# B&R Automation Studio project PrzewijarkaBRPraktyki
Automation Studio 4.12.8.41 SP; technology packages: mapp 5.24.5, mappCockpit 5.24.4, mappControl 5.24.2, mappMotion 5.29.0, mappView 5.24.5

## Configuration PrzewijarkaPraktykiBR

CPU X20CP0483, AutomationRuntime J4.93, Build 4.1.2, Safety 0.0, Vc V4.73.2

### Task classes (Cpu.sw)
```
Cyclic#4 (cycle 100000 us, tolerance 100000 us):
  PID <- Control.PID.PID.prg
  Tension <- Control.Tension.Tension.prg
  Axis1 <- Control.Axis.Axis1.Axis1.prg
  Axis2 <- Control.Axis.Axis2.Axis2.prg
  Axis3 <- Control.Axis.Axis3.Axis3.prg
  Axes <- Control.Axis.Axes.prg
  PackML <- PackMLCore.PackML.prg
NcDataObjects: mcdrivelog
Binaries: Settings, arcoal, mvLoader, arsvcreg, FWRules, arflatprv, udbdef, mCoWebSc, TCData, arconfig, User, sysconf, Role, iomap, asfw, ashwac, ashwd
Libraries: McBase, MpBase, sys_lib, arssl, MpAxis, McAxis, McAcpAx, MpAlarmX, astime, runtime, MpServer, CoTrace, AsZip, FileIO, MpRegMark, MpTension, MpPackML
```

### Hardware
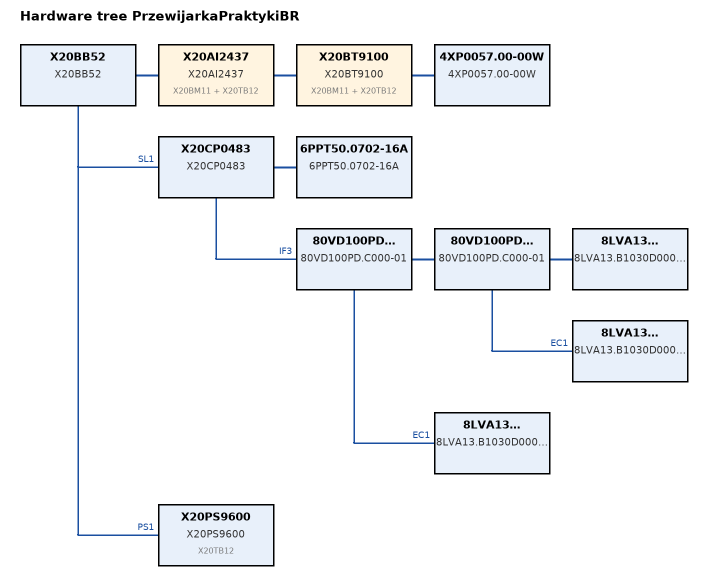
```
4XP0057.00-00W : 4XP0057.00-00W v2.1.0.0  [X2X1 -> X20BT9100.X2X1 [Cable Type=X2XCable, Length=10, Version=1.0.0.3]]
6PPT50.0702-16A : 6PPT50.0702-16A v1.3.8.0  [ETH1 -> X20CP0483.IF2 [Cable Type=PowerlinkCable, Length=10, Version=1.0.0.3]]
  Terminal = true
  Startmode = 2
  Mode = Manual
  InternetAddress = 192.168.0.12
  Subnetmask = 255.255.255.0
  PasswordVNC = 
  SelectedFavoriteWeb = 192.168.0.2
  Favorites_Web1 = webserver1
  PasswordCIFS = 
  PasswordService = 
80VD100PD.C000-01 : 80VD100PD.C000-01 v2.5.0.0  [PLK1 -> X20CP0483.IF3 (NodeNumber=1) [Cable Type=PowerlinkCable, Length=10, Version=1.0.0.3]; PLK2 -> 80VD100PD.C000-01a.PLK1 (NodeNumber=1) [Cable Type=PowerlinkCable, Length=10, Version=1.0.0.3]; EC1 -> 8LVA13.B1030D000-0.EC]
  DriveConfiguration/Module:
    McAcoposTypeID = AcoposMicroDConfig
    ActivateACOPOSSimulationOnPLC = 0
  DriveConfiguration/Channel[1]/RealAxis:
    AxisReference = gAxis_1
    MechanicalElementsIsInvisible = 0
  DriveConfiguration/Channel[1]/RealAxis/MechanicalElements/Gearbox:
    InputIsReadOnly = 0
    Input = 3
    OutputIsReadOnly = 0
    Output = 1
  DriveConfiguration/Channel[1]/RealAxis/MechanicalElements/RotaryToLinearTransformation:
    ReferenceDistanceIsReadOnly = 0
    ReferenceDistance = 360
  DriveConfiguration/Channel[1]/RealAxis/Controller:
    ModeIsReadOnly = 0
    Mode = PositionController
  DriveConfiguration/Channel[1]/RealAxis/Controller/Mode/Position:
    ProportionalGain = 358.000000
    IntegrationTime = 0.0
    PredictionTime = 0.0004
    TotalDelayTime = 0.0004
  DriveConfiguration/Channel[1]/RealAxis/Controller/Mode/Speed:
    ProportionalGainIsReadOnly = 0
    ProportionalGain = 1.150000
    IntegrationTimeIsReadOnly = 0
    IntegrationTime = 0.0
    FilterTimeIsReadOnly = 0
    FilterTime = 0.0
  DriveConfiguration/Channel[1]/RealAxis/Controller/Mode/LoopFilters:
    LoopFilterXIsReadOnly = 0
    LoopFilter1 = NotUsed
    LoopFilter2 = NotUsed
    LoopFilter3 = NotUsed
  DriveConfiguration/Channel[1]/RealAxis/Homing:
    ModeIsReadOnly = 0
    Mode = Direct
  DriveConfiguration/Channel[1]/RealAxis/Homing/Mode:
    Position = 0.0
    ReferencePulse = NotUsed
  DriveConfiguration/Channel[1]/RealAxis/Homing:
    RestorePositionVariable = 
  DriveConfiguration/Channel[1]/RealAxis/StopReaction:
    QuickstopIsReadOnly = 0
    Quickstop = DecelerationLimit
    DriveErrorIsReadOnly = 0
    DriveError = DecelerationLimit
    FilterTime = 0.0
  DriveConfiguration/Channel[1]/RealAxis/MovementErrorLimits:
    PositionError = 1.0
    VelocityErrorMonitoring = Automatic1
  DriveConfiguration/Channel[1]/RealAxis:
    JerkFilterIsReadOnly = 0
    JerkFilter = NotUsed
    ZeroVibrationFilter = NotUsed
  DriveConfiguration/Channel[1]/RealAxis/DigitalInputs/HomingSwitch:
    SourceIsReadOnly = 0
    Source = NotUsed
    Level = High
  DriveConfiguration/Channel[1]/RealAxis/DigitalInputs/PositiveLimitSwitch:
    SourceIsReadOnly = 0
    Source = NotUsed
    Level = High
  DriveConfiguration/Channel[1]/RealAxis/DigitalInputs/NegativeLimitSwitch:
    SourceIsReadOnly = 0
    Source = NotUsed
    Level = High
  DriveConfiguration/Channel[1]/RealAxis/DigitalInputs/Trigger1:
    Source = X2Trigger1
    Level = High
  DriveConfiguration/Channel[1]/RealAxis/DigitalInputs/Trigger2:
    Source = X2Trigger2
    Level = High
  DriveConfiguration/Channel[1]/RealAxis/DigitalInputs/Quickstop:
    Input = Trigger2
  DriveConfiguration/Channel[1]/RealAxis/Simulation:
    SimulationModeOnPLC = SetValueGeneration
    SimulationModeOnACOPOS = NotUsed
  DriveConfiguration/Channel[1]:
    ExternalEncoderAxis = NotUsed
  DriveConfiguration/Channel[2]/RealAxis:
    AxisReference = 
    MechanicalElementsIsInvisible = 0
  DriveConfiguration/Channel[2]/RealAxis/MechanicalElements/Gearbox:
    InputIsReadOnly = 0
    Input = 1
    OutputIsReadOnly = 0
    Output = 1
  DriveConfiguration/Channel[2]/RealAxis/MechanicalElements/RotaryToLinearTransformation:
    ReferenceDistanceIsReadOnly = 0
    ReferenceDistance = 1
  DriveConfiguration/Channel[2]/RealAxis/Controller:
    ModeIsReadOnly = 0
    Mode = PositionController
  DriveConfiguration/Channel[2]/RealAxis/Controller/Mode/Position:
    ProportionalGain = 50.0
    IntegrationTime = 0.0
    PredictionTime = 0.0004
    TotalDelayTime = 0.0004
  DriveConfiguration/Channel[2]/RealAxis/Controller/Mode/Speed:
    ProportionalGainIsReadOnly = 0
    ProportionalGain = 2.0
    IntegrationTimeIsReadOnly = 0
    IntegrationTime = 0.0
    FilterTimeIsReadOnly = 0
    FilterTime = 0.0
  DriveConfiguration/Channel[2]/RealAxis/Controller/Mode/LoopFilters:
    LoopFilterXIsReadOnly = 0
    LoopFilter1 = NotUsed
    LoopFilter2 = NotUsed
    LoopFilter3 = NotUsed
  DriveConfiguration/Channel[2]/RealAxis/Homing:
    ModeIsReadOnly = 0
    Mode = Direct
  DriveConfiguration/Channel[2]/RealAxis/Homing/Mode:
    Position = 0.0
    ReferencePulse = NotUsed
  DriveConfiguration/Channel[2]/RealAxis/Homing:
    RestorePositionVariable = 
  DriveConfiguration/Channel[2]/RealAxis/StopReaction:
    QuickstopIsReadOnly = 0
    Quickstop = DecelerationLimit
    DriveErrorIsReadOnly = 0
    DriveError = DecelerationLimit
    FilterTime = 0.0
  DriveConfiguration/Channel[2]/RealAxis/MovementErrorLimits:
    PositionError = 1.0
    VelocityErrorMonitoring = Automatic1
  DriveConfiguration/Channel[2]/RealAxis:
    JerkFilterIsReadOnly = 0
    JerkFilter = NotUsed
    ZeroVibrationFilter = NotUsed
  DriveConfiguration/Channel[2]/RealAxis/DigitalInputs/HomingSwitch:
    SourceIsReadOnly = 0
    Source = NotUsed
    Level = High
  DriveConfiguration/Channel[2]/RealAxis/DigitalInputs/PositiveLimitSwitch:
    SourceIsReadOnly = 0
    Source = NotUsed
    Level = High
  DriveConfiguration/Channel[2]/RealAxis/DigitalInputs/NegativeLimitSwitch:
    SourceIsReadOnly = 0
    Source = NotUsed
    Level = High
  DriveConfiguration/Channel[2]/RealAxis/DigitalInputs/Trigger1:
    Source = X2Trigger1
    Level = High
  DriveConfiguration/Channel[2]/RealAxis/DigitalInputs/Trigger2:
    Source = X2Trigger2
    Level = High
  DriveConfiguration/Channel[2]/RealAxis/DigitalInputs/Quickstop:
    Input = Trigger2
  DriveConfiguration/Channel[2]/RealAxis/Simulation:
    SimulationModeOnPLC = SetValueGeneration
    SimulationModeOnACOPOS = NotUsed
  DriveConfiguration/Channel[2]:
    ExternalEncoderAxis = NotUsed
80VD100PD.C000-01a : 80VD100PD.C000-01 v2.5.0.0  [PLK1 -> 80VD100PD.C000-01.PLK2 (NodeNumber=2) [Cable Type=PowerlinkCable, Length=10, Version=1.0.0.3]; EC1 -> 8LVA13.B1030D000-0b.EC; EC2 -> 8LVA13.B1030D000-0a.EC; MT2 -> 8LVA13.B1030D000-0a.MT]
  DriveConfiguration/Module:
    McAcoposTypeID = AcoposMicroDConfig
    ActivateACOPOSSimulationOnPLC = 0
  DriveConfiguration/Channel[1]/RealAxis:
    AxisReference = gAxis_2
    MechanicalElementsIsInvisible = 0
  DriveConfiguration/Channel[1]/RealAxis/MechanicalElements/Gearbox:
    InputIsReadOnly = 0
    Input = 3
    OutputIsReadOnly = 0
    Output = 1
  DriveConfiguration/Channel[1]/RealAxis/MechanicalElements/RotaryToLinearTransformation:
    ReferenceDistanceIsReadOnly = 0
    ReferenceDistance = 191.637
  DriveConfiguration/Channel[1]/RealAxis/Controller:
    ModeIsReadOnly = 0
    Mode = PositionController
  DriveConfiguration/Channel[1]/RealAxis/Controller/Mode/Position:
    ProportionalGain = 124.000000
    IntegrationTime = 0.0
    PredictionTime = 0.0004
    TotalDelayTime = 0.0004
  DriveConfiguration/Channel[1]/RealAxis/Controller/Mode/Speed:
    ProportionalGainIsReadOnly = 0
    ProportionalGain = 0.950000
    IntegrationTimeIsReadOnly = 0
    IntegrationTime = 0.0
    FilterTimeIsReadOnly = 0
    FilterTime = 0.0
  DriveConfiguration/Channel[1]/RealAxis/Controller/Mode/LoopFilters:
    LoopFilterXIsReadOnly = 0
    LoopFilter1 = NotUsed
    LoopFilter2 = NotUsed
    LoopFilter3 = NotUsed
  DriveConfiguration/Channel[1]/RealAxis/Homing:
    ModeIsReadOnly = 0
    Mode = Direct
  DriveConfiguration/Channel[1]/RealAxis/Homing/Mode:
    Position = 0.0
    ReferencePulse = NotUsed
  DriveConfiguration/Channel[1]/RealAxis/Homing:
    RestorePositionVariable = 
  DriveConfiguration/Channel[1]/RealAxis/StopReaction:
    QuickstopIsReadOnly = 0
    Quickstop = DecelerationLimit
    DriveErrorIsReadOnly = 0
    DriveError = DecelerationLimit
    FilterTime = 0.0
  DriveConfiguration/Channel[1]/RealAxis/MovementErrorLimits:
    PositionError = 1.0
    VelocityErrorMonitoring = Automatic1
  DriveConfiguration/Channel[1]/RealAxis:
    JerkFilterIsReadOnly = 0
    JerkFilter = NotUsed
    ZeroVibrationFilter = NotUsed
  DriveConfiguration/Channel[1]/RealAxis/DigitalInputs/HomingSwitch:
    SourceIsReadOnly = 0
    Source = NotUsed
    Level = High
  DriveConfiguration/Channel[1]/RealAxis/DigitalInputs/PositiveLimitSwitch:
    SourceIsReadOnly = 0
    Source = NotUsed
    Level = High
  DriveConfiguration/Channel[1]/RealAxis/DigitalInputs/NegativeLimitSwitch:
    SourceIsReadOnly = 0
    Source = NotUsed
    Level = High
  DriveConfiguration/Channel[1]/RealAxis/DigitalInputs/Trigger1:
    Source = X2Trigger1
    Level = High
  DriveConfiguration/Channel[1]/RealAxis/DigitalInputs/Trigger2:
    Source = X2Trigger2
    Level = High
  DriveConfiguration/Channel[1]/RealAxis/DigitalInputs/Quickstop:
    Input = Trigger2
  DriveConfiguration/Channel[1]/RealAxis/Simulation:
    SimulationModeOnPLC = SetValueGeneration
    SimulationModeOnACOPOS = NotUsed
  DriveConfiguration/Channel[1]:
    VirtualAxis = Used
  DriveConfiguration/Channel[1]/VirtualAxis:
    AxisReference = 
  DriveConfiguration/Channel[1]/VirtualAxis/Homing:
    Mode = Direct
  DriveConfiguration/Channel[1]/VirtualAxis/Homing/Mode:
    Position = 0.0
  DriveConfiguration/Channel[1]/VirtualAxis/Homing:
    RestorePositionVariable = 
  DriveConfiguration/Channel[1]/VirtualAxis:
    JerkFilterIsReadOnly = 0
    JerkFilter = NotUsed
    ZeroVibrationFilter = NotUsed
  DriveConfiguration/Channel[1]:
    ExternalEncoderAxis = NotUsed
  DriveConfiguration/Channel[2]/RealAxis:
    AxisReference = gAxis_3
    MechanicalElementsIsInvisible = 0
  DriveConfiguration/Channel[2]/RealAxis/MechanicalElements/Gearbox:
    InputIsReadOnly = 0
    Input = 3
    OutputIsReadOnly = 0
    Output = 1
  DriveConfiguration/Channel[2]/RealAxis/MechanicalElements/RotaryToLinearTransformation:
    ReferenceDistanceIsReadOnly = 0
    ReferenceDistance = 360
  DriveConfiguration/Channel[2]/RealAxis/Controller:
    ModeIsReadOnly = 0
    Mode = PositionController
  DriveConfiguration/Channel[2]/RealAxis/Controller/Mode/Position:
    ProportionalGain = 358
    IntegrationTime = 0.0
    PredictionTime = 0.0004
    TotalDelayTime = 0.0004
  DriveConfiguration/Channel[2]/RealAxis/Controller/Mode/Speed:
    ProportionalGainIsReadOnly = 0
    ProportionalGain = 1.15
    IntegrationTimeIsReadOnly = 0
    IntegrationTime = 0.0
    FilterTimeIsReadOnly = 0
    FilterTime = 0.0
  DriveConfiguration/Channel[2]/RealAxis/Controller/Mode/LoopFilters:
    LoopFilterXIsReadOnly = 0
    LoopFilter1 = NotUsed
    LoopFilter2 = NotUsed
    LoopFilter3 = NotUsed
  DriveConfiguration/Channel[2]/RealAxis/Homing:
    ModeIsReadOnly = 0
    Mode = Direct
  DriveConfiguration/Channel[2]/RealAxis/Homing/Mode:
    Position = 0.0
    ReferencePulse = NotUsed
  DriveConfiguration/Channel[2]/RealAxis/Homing:
    RestorePositionVariable = 
  DriveConfiguration/Channel[2]/RealAxis/StopReaction:
    QuickstopIsReadOnly = 0
    Quickstop = DecelerationLimit
    DriveErrorIsReadOnly = 0
    DriveError = DecelerationLimit
    FilterTime = 0.0
  DriveConfiguration/Channel[2]/RealAxis/MovementErrorLimits:
    PositionError = 1.0
    VelocityErrorMonitoring = Automatic1
  DriveConfiguration/Channel[2]/RealAxis:
    JerkFilterIsReadOnly = 0
    JerkFilter = NotUsed
    ZeroVibrationFilter = NotUsed
  DriveConfiguration/Channel[2]/RealAxis/DigitalInputs/HomingSwitch:
    SourceIsReadOnly = 0
    Source = NotUsed
    Level = High
  DriveConfiguration/Channel[2]/RealAxis/DigitalInputs/PositiveLimitSwitch:
    SourceIsReadOnly = 0
    Source = NotUsed
    Level = High
  DriveConfiguration/Channel[2]/RealAxis/DigitalInputs/NegativeLimitSwitch:
    SourceIsReadOnly = 0
    Source = NotUsed
    Level = High
  DriveConfiguration/Channel[2]/RealAxis/DigitalInputs/Trigger1:
    Source = X2Trigger1
    Level = High
  DriveConfiguration/Channel[2]/RealAxis/DigitalInputs/Trigger2:
    Source = X2Trigger2
    Level = High
  DriveConfiguration/Channel[2]/RealAxis/DigitalInputs/Quickstop:
    Input = Trigger2
  DriveConfiguration/Channel[2]/RealAxis/Simulation:
    SimulationModeOnPLC = SetValueGeneration
    SimulationModeOnACOPOS = NotUsed
  DriveConfiguration/Channel[2]:
    ExternalEncoderAxis = NotUsed
8LVA13.B1030D000-0 : 8LVA13.B1030D000-0 v2.2.0.3  [EC -> 80VD100PD.C000-01.EC1; MT -> 80VD100PD.C000-01.MT1]
  M1/MotorParameters:
    MOTOR_AMB_TEMP_RATED = 40
8LVA13.B1030D000-0a : 8LVA13.B1030D000-0 v2.2.0.3  [EC -> 80VD100PD.C000-01a.EC2; MT -> 80VD100PD.C000-01a.MT2]
  M1/MotorParameters:
    MOTOR_AMB_TEMP_RATED = 40
8LVA13.B1030D000-0b : 8LVA13.B1030D000-0 v2.2.0.3  [EC -> 80VD100PD.C000-01a.EC1; MT -> 80VD100PD.C000-01a.MT1]
  M1/MotorParameters:
    MOTOR_AMB_TEMP_RATED = 40
X20AI2437 : X20AI2437 v1.3.0.0  [SS1 -> X20TB12a.SS; SL -> X20BM11.SL1]
X20BB52 : X20BB52 v1.2.0.0
X20BM11 : X20BM11 v1.1.0.0  [X2X1 -> X20BB52.IF6]
X20BM11a : X20BM11 v1.1.0.0  [X2X1 -> X20BM11.X2X2]
X20BT9100 : X20BT9100 v1.3.0.0  [SS1 -> X20TB12b.SS; SL -> X20BM11a.SL1]
X20CP0483 : X20CP0483 v1.6.0.0  [SL -> X20BB52.SL1]
  Connector IF2:
    ActivateDevice = 1
    Mode = Manual
    InternetAddress = 192.168.0.2
    SubnetMask = 255.255.255.0
  Connector IF3:
    Channel1
    ChannelID1 = McAcpBroadcast
    ChannelType1 = OCTET[36]
  ConfigurationID = PrzewijarkaBRPraktyki_PrzewijarkaPraktykiBR
  TimerDeviceType = EPLX2X
  TimerDevice = X20CP0483.IF3
  TaskClassIdleTime = 2000
  Cyclic1Duration = 2000
  Cyclic1Tolerance = 0
  Cyclic1Stack = 30000
  Cyclic1Output = 1
  Cyclic2Duration = 20000
  Cyclic2Tolerance = 20000
  Cyclic3Duration = 50000
  Cyclic3Tolerance = 50000
  Cyclic4Duration = 100000
  Cyclic4Tolerance = 100000
  Cyclic5Duration = 200000
  Cyclic5Tolerance = 200000
  Cyclic6Duration = 500000
  Cyclic6Tolerance = 500000
  Cyclic7Duration = 1000000
  Cyclic7Tolerance = 1000000
  Cyclic8Duration = 10000
  Cyclic8Tolerance = 30000000
  FileDevice1
  FileDeviceName1 = USER
  FileDevicePath1 = USER_PATH
  FileDevice2
  FileDeviceName2 = RECIPE
  FileDevicePath2 = USER_PATH/Recipe
  FileDevice3
  FileDeviceName3 = DATA
  FileDevicePath3 = USER_PATH/Data
  TimeZone = 160
  ActivateDaylightSavingTime = 1
  ActivateSntpServer = 1
  EthernetDefaultGateway = 192.168.0.1
  FtpUser1
  FtpUsername1 = AdminFTP
  FtpUserPassword1 = 6YI7hPEHEUgPCGBGJ1BSV9dcZzKYXQvWVp6sNHSerZA=  // Admin123
  FtpUserSalt1 = /B0I6o9l
  FTPAccessRight1 = 0
  ActivateOpcUa = 1
  OpcUaInformationModels_PV_Version = 1
X20PS9600 : X20PS9600 v1.6.0.0  [PS -> X20BB52.PS1; SS1 -> X20TB12.SS]
X20TB12 : X20TB12 v1.0.0.0
X20TB12a : X20TB12 v1.0.0.0
X20TB12b : X20TB12 v1.0.0.0
```

### IoMap.iom - X20CP0483/IoMap.iom
```iecst
VAR_CONFIG
	::gHMI.ModuleOK.PowerSupply AT %IX."X20PS9600".ModuleOk;
	::gHMI.ModuleOK.AnalogInput AT %IX."X20AI2437".ModuleOk;
	::gHMI.ModuleOK.SystemBusTransmitter AT %IX."X20BT9100".ModuleOk;
	::gHMI.ModuleOK.ControlKeypad AT %IX."4XP0057.00-00W".ModuleOk;
	::Tension:ActRightDancerPos AT %IW."X20AI2437".AnalogInput01;
	::Tension:ActLeftDancerPos AT %IW."X20AI2437".AnalogInput02;
	::MainPage:PhysicalBtn.Production.Start.State AT %IX."4XP0057.00-00W".DigitalInput01;
	::MainPage:PhysicalBtn.Production.Stop.State AT %IX."4XP0057.00-00W".DigitalInput02;
	::MainPage:PhysicalBtn.Production.Reset.State AT %IX."4XP0057.00-00W".DigitalInput05;
	::MainPage:PhysicalBtn.Manual.Left.State AT %IX."4XP0057.00-00W".DigitalInput03;
	::MainPage:PhysicalBtn.Manual.Right.State AT %IX."4XP0057.00-00W".DigitalInput04;
	::MainPage:PhysicalBtn.Production.Start.ColorON AT %QX."4XP0057.00-00W".DigitalOutput01;
	::MainPage:PhysicalBtn.Production.Stop.ColorON AT %QX."4XP0057.00-00W".DigitalOutput07;
	::MainPage:PhysicalBtn.Manual.Left.ColorON AT %QX."4XP0057.00-00W".DigitalOutput12;
	::MainPage:PhysicalBtn.Manual.Right.ColorON AT %QX."4XP0057.00-00W".DigitalOutput16;
	::MainPage:PhysicalBtn.Production.Reset.ColorON AT %QX."4XP0057.00-00W".DigitalOutput20;
END_VAR
```

### Config_2.tensioncontroller - X20CP0483/mappControl/Config_2.tensioncontroller
```
Element gTensionCtrl_Unwinder (Type=tensioncontroller)  // axis1
  TensionController:
    MotionSystem = mappMotion
      AxisReference = gAxis_1
      AxisVelocityProfile:
        Acceleration = 0.5
        Deceleration = 0.5
        StopDeceleration = 2
    Utilization:
      Winder:
        MinimumDiameter = 30
        MaximumDiameter = 80
    Controller:
      PIDParameters:
        OperatingPoint[1]
      MaximumVelocityCorrection = 1
      ToleranceBand:
        Lower = 4
        Upper = 4
      Initialization:
        MaximumLineVelocityCorrection = 1
    Material:
      Length = 0.4
      Width = 48
      TensionLimit = 300
    InputSignals:
      SetMaterialTension = 
Element gTensionCtrl_Rewinder (Type=tensioncontroller)  // axis3
  TensionController:
    MotionSystem = mappMotion
      AxisReference = gAxis_3
      AxisVelocityProfile:
        Acceleration = 0.5
        Deceleration = 0.5
        StopDeceleration = 2
    Utilization = Rewind
      Winder:
        MinimumDiameter = 30
        MaximumDiameter = 80
    Controller:
      PIDParameters:
        OperatingPoint[1]
      ToleranceBand:
        Lower = 4
        Upper = 4
      Initialization:
        MaximumLineVelocityCorrection = 1
    Material:
      Length = 0.4
      Width = 48
      TensionLimit = 300
    InputSignals:
      SetMaterialTension = 
Element gTensionCtrl_Master (Type=tensioncontroller)
  TensionController:
    Utilization = Transport
    Controller = Master
Element gTensionCtrl_TransportDancer (Type=tensioncontroller)  // axis2
  TensionController:
    MotionSystem = mappMotion
      AxisReference = gAxis_2
      AxisVelocityProfile:
        Acceleration = 0.5
        Deceleration = 0.5
        StopDeceleration = 2
    Utilization = Transport
    Controller = DancerControl
      PIDParameters:
        OperatingPoint[1]
      Orientation = 1
      Initialization:
        MaximumLineVelocityCorrection = 1
    Material:
      Length = 0.4
      TensionLimit = 300
    InputSignals:
      SetDancerPosition = 
Element gTensionCtrl_TransportTension (Type=tensioncontroller)
  TensionController:
    Utilization = Transport
    Controller:
      PIDParameters:
        OperatingPoint[1]
```

### Config_3.tensiongroup - X20CP0483/mappControl/Config_3.tensiongroup
```
Element gTensionGroup_1 (Type=tensiongroup)
  Linking:
    Subnodes:
      Zone[0] = gTensionCtrl_Unwinder
      Zone[1] = gTensionCtrl_TransportDancer
      Zone[2] = gTensionCtrl_Rewinder
  TensionGroup:
    Simulation = 1
    CommonZoneSettings:
      Material:
        Width = 48
        TensionLimit = 300
    InputSignals:
      GroupLineVelocity = ::Tension:TensionVar.GroupLineVelocity
    Features:
      FeatureRef[0] = 
```

### Config_4.regmarkdetection - X20CP0483/mappControl/Config_4.regmarkdetection
```
Element gRegMarkDetection_1 (Type=regmarkdetection)
  RegistrationMarkDetection:
    SensorSignal:
      AxisReference = gAxis_2
```

### Config_8.purevaxcfg - X20CP0483/mappMotion/Config_8.purevaxcfg
```
Element PureVAxCfg_1 (Type=purevaxcfg)
  TypeID = PureVAxConfig
  PureVAxis:
    AxisReference = gAxisMaster
    Homing:
      Mode = Direct
        Position = 0.0
        ReferencePulse = NotUsed
      RestorePositionVariable
    JerkFilter = NotUsed
    ZeroVibrationFilter = NotUsed
    GeneralPurposeAxisInterface = Used
      Module:
        ActivateModuleSimulationOnPLC = Off
      MechanicalElements:
        Gearbox:
          InputIsReadOnly = 0
          Input = 3
          OutputIsReadOnly = 0
          Output = 1
        RotaryToLinearTransformation:
          ReferenceDistanceIsReadOnly = 0
          ReferenceDistance = 0.195
      EncoderLink = NoEncoder
      Controller:
        ModeIsReadOnly = 0
        Mode = PositionController
          Position:
            ProportionalGain = 124.000000
            IntegrationTime = 0.0
            PredictionTime = 0.0004
            TotalDelayTime = 0.0004
            MaximumProportionalAction = 1e30
            MaximumIntegralAction = 0.0
      StopReaction:
        Quickstop = DecelerationLimit
        DriveError = DecelerationLimit
      MovementErrorLimits:
        PositionError = 0.0
      DigitalInputs:
        HomingSwitch:
          Source = NotUsed
          Level = High
        PositiveLimitSwitch:
          Source = NotUsed
          Level = High
        NegativeLimitSwitch:
          Source = NotUsed
          Level = High
        Trigger1:
          Source = NotUsed
          Level = High
        Trigger2:
          Source = NotUsed
          Level = High
        Quickstop:
          Input = NotUsed
      StatusInputs:
        PoweredOn:
          Source = NotUsed
        CommunicationReady:
          Source = NotUsed
        ReadyForPowerOn:
          Source = NotUsed
        ErrorReactionActive:
          Source = NotUsed
        Error:
          Source = NotUsed
        ErrorID:
          Source = NotUsed
        Warning:
          Source = NotUsed
        WarningID:
          Source = NotUsed
      ControlOutputs:
        PowerOn = NotUsed
        ErrorReset = NotUsed
        BrakeControl = NotUsed
        SetSpeed = NotUsed
        SetPosition = NotUsed
      Simulation:
        LoadSimulationMode = NotUsed
```

### MotorLeft.axis - X20CP0483/mappMotion/MotorLeft.axis
```
Element gAxis_1 (Type=axis)
  BaseTypeIsReadOnly = 0
  BaseType = Rotary
    MeasurementUnitIsReadOnly = 0
    MeasurementUnit = 17476
    MeasurementResolutionIsReadOnly = 0
    MeasurementResolution = 0.01
    CountDirectionIsReadOnly = 0
    CountDirection = Standard
  MovementLimitsIsReadOnly = 0
  MovementLimits = Internal
    Position:
      LowerLimitMin = -1.79769313486231E308
      UpperLimitMax = 1.79769313486231E308
      LowerLimit = -1000.0
      UpperLimit = 1000.0
    VelocityIsReadOnly = 0
    Velocity:
      VelocityMax = 3.4E38
      Velocity = 100000
    AccelerationIsReadOnly = 0
    Acceleration:
      AccelerationMax = 3.4E38
      Acceleration = 50000.0
    DecelerationIsReadOnly = 0
    Deceleration:
      DecelerationMax = 3.4E38
      Deceleration = 50000.0
  Alarms = MpAlarmX
```

### MotorMid.axis - X20CP0483/mappMotion/MotorMid.axis
```
Element gAxis_2 (Type=axis)
  BaseTypeIsReadOnly = 0
  BaseType = Linear
    MeasurementUnit = 5066068
    MeasurementResolutionIsReadOnly = 0
    MeasurementResolution = 0.01
    CountDirectionIsReadOnly = 0
    CountDirection = Inverse
  MovementLimitsIsReadOnly = 0
  MovementLimits = Internal
    Position:
      LowerLimitMin = -1.79769313486231E308
      UpperLimitMax = 1.79769313486231E308
      LowerLimit = -1000.0
      UpperLimit = 1000.0
    VelocityIsReadOnly = 0
    Velocity:
      VelocityMax = 3.4E38
      Velocity = 10000.0
    AccelerationIsReadOnly = 0
    Acceleration:
      AccelerationMax = 3.4E38
      Acceleration = 100000.0
    DecelerationIsReadOnly = 0
    Deceleration:
      DecelerationMax = 3.4E38
      Deceleration = 100000.0
  Alarms = MpAlarmX
```

### MotorRight.axis - X20CP0483/mappMotion/MotorRight.axis
```
Element gAxis_3 (Type=axis)
  BaseTypeIsReadOnly = 0
  BaseType = Rotary
    MeasurementUnitIsReadOnly = 0
    MeasurementUnit = 17476
    MeasurementResolutionIsReadOnly = 0
    MeasurementResolution = 0.01
    CountDirectionIsReadOnly = 0
    CountDirection = Standard
  MovementLimitsIsReadOnly = 0
  MovementLimits = Internal
    Position:
      LowerLimitMin = -1.79769313486231E308
      UpperLimitMax = 1.79769313486231E308
      LowerLimit = -1000.0
      UpperLimit = 1000.0
    VelocityIsReadOnly = 0
    Velocity:
      VelocityMax = 3.4E38
      Velocity = 100000
    AccelerationIsReadOnly = 0
    Acceleration:
      AccelerationMax = 3.4E38
      Acceleration = 50000.0
    DecelerationIsReadOnly = 0
    Deceleration:
      DecelerationMax = 3.4E38
      Deceleration = 50000.0
  Alarms = MpAlarmX
```

### PureVAxis.axis - X20CP0483/mappMotion/PureVAxis.axis
```
Element gAxisMaster (Type=axis)
  BaseTypeIsReadOnly = 0
  BaseType = Linear
    MeasurementUnit = 5066068
    MeasurementResolutionIsReadOnly = 0
    MeasurementResolution = 0.01
    CountDirectionIsReadOnly = 0
    CountDirection = Standard
  MovementLimitsIsReadOnly = 0
  MovementLimits = Internal
    Position:
      LowerLimitMin = -1.79769313486231E308
      UpperLimitMax = 1.79769313486231E308
      LowerLimit = -1000.0
      UpperLimit = 1000.0
    VelocityIsReadOnly = 0
    Velocity:
      VelocityMax = 3.4E38
      Velocity = 10000
    AccelerationIsReadOnly = 0
    Acceleration:
      AccelerationMax = 3.4E38
      Acceleration = 200.0
    DecelerationIsReadOnly = 0
    Deceleration:
      DecelerationMax = 3.4E38
      Deceleration = 200.0
  Alarms = MpAlarmX
```

### VAxisConf.purevaxcfg - X20CP0483/mappMotion/VAxisConf.purevaxcfg
```
Element PureVAxCfg (Type=purevaxcfg)
  TypeID = PureVAxConfig
  PureVAxis:
    AxisReference = gAxisMaster
    Homing:
      Mode = Direct
        Position = 0.0
        ReferencePulse = NotUsed
      RestorePositionVariable
    JerkFilter = NotUsed
    ZeroVibrationFilter = NotUsed
    GeneralPurposeAxisInterface = Used
      Module:
        ActivateModuleSimulationOnPLC = On
      MechanicalElements:
        Gearbox:
          InputIsReadOnly = 0
          Input = 3
          OutputIsReadOnly = 0
          Output = 1
        RotaryToLinearTransformation:
          ReferenceDistanceIsReadOnly = 0
          ReferenceDistance = 0.195
      EncoderLink = NoEncoder
      Controller:
        ModeIsReadOnly = 0
        Mode = NotUsed
      StopReaction:
        Quickstop = DecelerationLimit
        DriveError = DecelerationLimit
      MovementErrorLimits:
        PositionError = 0.0
      DigitalInputs:
        HomingSwitch:
          Source = NotUsed
          Level = High
        PositiveLimitSwitch:
          Source = NotUsed
          Level = High
        NegativeLimitSwitch:
          Source = NotUsed
          Level = High
        Trigger1:
          Source = NotUsed
          Level = High
        Trigger2:
          Source = NotUsed
          Level = High
        Quickstop:
          Input = NotUsed
      StatusInputs:
        PoweredOn:
          Source = NotUsed
        CommunicationReady:
          Source = NotUsed
        ReadyForPowerOn:
          Source = NotUsed
        ErrorReactionActive:
          Source = NotUsed
        Error:
          Source = NotUsed
        ErrorID:
          Source = NotUsed
        Warning:
          Source = NotUsed
        WarningID:
          Source = NotUsed
      ControlOutputs:
        PowerOn = NotUsed
        ErrorReset = NotUsed
        BrakeControl = NotUsed
        SetSpeed = NotUsed
        SetPosition = NotUsed
      Simulation:
        LoadSimulationMode = SetValueGeneration
```

### Config.mpalarmxcore - X20CP0483/mappServices/Config.mpalarmxcore
```
Element gAlarmXCore (Type=mpalarmxcore)
  mapp.AlarmX.Core.Configuration:
    [0]:
      Name = ModuleOKErrorPS
      Message = Power supply module uninstalled, not present or broken
      Behavior = PersistentAlarm
    [1]:
      Name = ModuleOKErrorAI
      Message = Analog input module uninstalled, not present or broken
      Code = 1
      Behavior = PersistentAlarm
    [2]:
      Name = ModuleOKErrorBT
      Message = System bus transmitter module uninstalled, not present or broken
      Behavior = PersistentAlarm
    [3]:
      Name = ModuleOKError4XP
      Message = Control keypad module uninstalled, not present or broken
      Behavior = PersistentAlarm
    [4]:
      Name = LeftWinderDiameterLow
      Message = Left winder diameter too low! Check tape volume
      Behavior = PersistentAlarm
    [5]:
      Name = RightWinderDiameterLow
      Message = Right winder diameter too low! Check tape volume
      Behavior = PersistentAlarm
```

### Config.mppackmlcore - X20CP0483/mappServices/Config.mppackmlcore
```
Element gPackMLCore (Type=mppackmlcore)
  Modes:
    Mode[1]:
      ModeID = 1
      Name = Production
    Mode[2]:
      Name = Mode[3]
```

### Config_1.mpalarmxhistory - X20CP0483/mappServices/Config_1.mpalarmxhistory
```
Element gAlarmXHistory (Type=mpalarmxhistory)
  mapp.AlarmX.History:
    Memory:
      MemoryType = 3
```

### Config_4.mpuserx - X20CP0483/mappServices/Config_4.mpuserx
```
Element UserMgmtX (Type=mpuserx)
  Mgr:
    EditSameLevel = TRUE
  ServerSettings:
    Server:
      AdditionalUserData:
        [0] = mail
        [1] = telephoneNumber
  Users:
    DefUser#1:
      id = Admin
      name = Administrators
    DefUser#2:
      id = Anonymous
      name = Everyone
    DefUser#3:
      id = OperatorUser
      name = Operator
    DefUser#4:
      id = SupervisorUser
      name = Supervisor
  Groups:
    DefGroup#1:
      id = Administrators
      admin = TRUE
    DefGroup#2:
      id = Everyone
    DefGroup#3:
      id = Operator
    DefGroup#4:
      id = Supervisor
```

### Config_5.mpaudittrail - X20CP0483/mappServices/Config_5.mpaudittrail
```
Element gAuditTrail (Type=mpaudittrail)
  Audit:
    Events:
      [0] = 16
      [1] = 2
      [2] = 18
      [3] = 33
      [4] = 64
      [5] = 65
      [6] = 48
    Export:
      RawData = TRUE
      FileType = 2
  Alarms = MpAlarmX
```

### Config_6.mprecipexml - X20CP0483/mappServices/Config_6.mprecipexml
```
Element MpLinkRecipes (Type=mprecipexml)
  mapp.Recipe.Xml:
    Auditing = MpAudit
```

### Config_7.mpdatarecorder - X20CP0483/mappServices/Config_7.mpdatarecorder
```
Element gDataRecorder (Type=mpdatarecorder)
  DataRecorder:
    MaxNumberOfFiles = 3
    OverwriteOldestFile = TRUE
  Alarms = MpAlarmX
```

### Config_PML.mppackmlcore - X20CP0483/mappServices/Config_PML.mppackmlcore
```
Element gPackMLCore (Type=mppackmlcore)
  Modes:
    Mode[1]:
      ModeID = 1
      Name = Production
    Mode[2]:
      ModeID = 2
      Name = Mode[3]
```

## Logical view

Binary libraries used (declarations not repeated): operator, runtime, astime, AsIecCon, McBase, MpBase, MpAxis, McAxis, McAcpAx, MpAlarmX, MpServer, CoTrace, AsZip, FileIO, MpRegMark, MpTension 5.24.2, MpPackML 5.24.5

### Package Logical/Libraries - Global libraries

### PackML_IF.typ
```iecst
TYPE
	StatusType : 	STRUCT
		ModeCurrent : STRING[20];
		StateCurrent : STRING[20];
	END_STRUCT;
END_TYPE
```

### Program Logical/PackMLCore/PackML (IEC)

#### Code.st - Init, cyclic, exit code
```iecst
PROGRAM _INIT
	(* Insert code here *)
	MpPackMLCore_0(MpLink := ADR(gPackMLCore), Enable := TRUE);
END_PROGRAM

PROGRAM _CYCLIC
	(* Insert code here *)
	MpPackMLCore_0(MpLink := ADR(gPackMLCore), Enable := TRUE);
END_PROGRAM

PROGRAM _EXIT
	(* Insert code here *)
	 MpPackMLCore_0(MpLink := ADR(gPackMLCore), Enable := FALSE);
END_PROGRAM
```

#### Variables.var - Local variables
```iecst
VAR
	MpPackMLMode_0 : MpPackMLMode;
	MpPackMLMode_1 : MpPackMLMode;
	MpPackMLBasicUI_0 : MpPackMLBasicUI;
	prevBtn : BOOL := FALSE; (* poprzedni stan przycisku *)
	step : INT := 0; (* maszyna stanów *)
	MpPackMLCore_0 : MpPackMLCore;
END_VAR
```

#### actInterface.st
```iecst
ACTION actInterface:

END_ACTION
```

#### actGetStatus.st
```iecst
ACTION actGetStatus:

END_ACTION
```

#### actResetCommands.st
```iecst
ACTION actResetCommands:

END_ACTION
```

### gPackML.typ - not listed in the package file held
```iecst
TYPE
	StatusType : 	STRUCT
		ModeCurrent : STRING[20];
		StateCurrent : STRING[20];
	END_STRUCT;
END_TYPE
```

### gPackML.var - not listed in the package file held
```iecst
VAR
	Status : StatusType;
	MpPackMLBasicUIConnect : MpPackMLBasicUIConnectType;
END_VAR
```

### Variables.var - not listed in the package file held
```iecst
VAR
	MpPackMLCore_0 : MpPackMLCore;
END_VAR
```

### Program Logical/Control/Tension/Tension (IEC)

#### TensionTyp.typ - Local data types
```iecst
TYPE
	TESTstate :
		(
		INIT,
		POWER,
		ERROR,
		ERROR_RESET,
		HOME,
		WAIT_FOR_COMMAND,
		MOVE_ABSOLUTE,
		TEST
		);
END_TYPE
```

#### TensionVar.var - Local variables
```iecst
VAR RETAIN
	RightWinderDiameter : REAL := 30.0;
	LeftWinderDiameter : REAL := 80.0;
END_VAR
VAR
	Step : StepEnum;
	PackMLMode : PackMLModes;
	TensionGroup : MpTensionGroup;
END_VAR
VAR CONSTANT
	NR_OF_ZONES : USINT := 3;
	INDEX_NR_OF_ZONES : USINT := NR_OF_ZONES-1;
END_VAR
VAR
	i : USINT;
	TensionController : ARRAY[0..INDEX_NR_OF_ZONES] OF MpTensionController;
	ActLeftDancerPos : INT;
	ActLeftDancerPosScal : REAL;
	Distance : REAL;
	SetRightDancerPos : REAL := 0.0;
	SetLeftDancerPos : REAL := 0.0;
	ActRightDancerPosScal : REAL;
	ProgressBarProcent : REAL;
	MpAxisBasicParams : ARRAY[0..2] OF MpAxisBasicParType;
	MpAxisBasicFB : ARRAY[0..2] OF MpAxisBasic;
	ActRightDancerPos : INT;
	StartingMaterialToProcess : REAL := 0.0;
END_VAR
```

#### TensionGroup.st - Init, cyclic, exit code
```iecst
PROGRAM _INIT
	actInitTension;
END_PROGRAM

PROGRAM _CYCLIC
	actReadGlobals;
	actLineInGroupVelocity;
	actDoAlgebra;
	actCallBlocks;
	actSetGlogals;
END_PROGRAM

PROGRAM _EXIT
    actExitTension;
END_PROGRAM
```

#### actInitTension.st
```iecst
ACTION actInitTension:
	gAxis_1;
	gAxis_2;
	gAxis_3;

	TensionController[0].MpLink := ADR(gTensionCtrl_Unwinder);
	TensionController[1].MpLink := ADR(gTensionCtrl_Master);
	TensionController[2].MpLink := ADR(gTensionCtrl_Rewinder);
	TensionGroup.MpLink := ADR(gTensionGroup_1);

	FOR i := 0 TO INDEX_NR_OF_ZONES DO

		TensionController[i].Enable := TRUE;
		MpAxisBasicFB[i].Enable := TRUE;

	END_FOR;

	TensionController[0].PresetDiameter := LeftWinderDiameter;
	TensionController[2].PresetDiameter := RightWinderDiameter;
	TensionController[0].SetPresetDiameter := TRUE;
	TensionController[2].SetPresetDiameter := TRUE;
	TensionGroup.Enable := TRUE;
	MpAxisBasicFB[0].MpLink := ADR(gAxis_1);
	MpAxisBasicFB[1].MpLink := ADR(gAxis_2);
	MpAxisBasicFB[2].MpLink := ADR(gAxis_3);

	MpAxisBasicFB[0].Parameters := ADR(MpAxisBasicParams[0]);
	MpAxisBasicFB[1].Parameters := ADR(MpAxisBasicParams[1]);
	MpAxisBasicFB[2].Parameters := ADR(MpAxisBasicParams[2]);

END_ACTION
```

#### actLineInGroupVelocity.st
```iecst
ACTION actLineInGroupVelocity:
	IF TensionGroup.InLineVelocity AND
		(((SetLeftDancerPos - 1) >= ActLeftDancerPosScal OR
		ActLeftDancerPosScal >= (SetLeftDancerPos + 1)) OR
		((SetRightDancerPos - 1) >= ActRightDancerPosScal OR
		ActRightDancerPosScal >= (SetRightDancerPos + 1))) THEN
		TensionGroup.Control := TRUE;
	ELSE
		TensionGroup.Control := FALSE;
	END_IF;
	IF (((SetLeftDancerPos - 1) >= ActLeftDancerPosScal OR
		ActLeftDancerPosScal >= (SetLeftDancerPos + 1)) OR
		((SetRightDancerPos - 1) >= ActRightDancerPosScal OR
		ActRightDancerPosScal >= (SetRightDancerPos + 1))) THEN
		gMainLogic.MotorMode.Production.Status.TensionReady := FALSE;
	ELSE
		gMainLogic.MotorMode.Production.Status.TensionReady := TRUE;
	END_IF;
END_ACTION
```

#### actDoAlgebra.st
```iecst
ACTION actDoAlgebra:
	ActLeftDancerPosScal :=  brmfloor(((INT_TO_REAL(ActLeftDancerPos) - 4060.0) *(1000.0/135534.0)));
	ActRightDancerPosScal := brmfloor(((INT_TO_REAL(ActRightDancerPos) - 4045.0) *(1000.0/135534.0)));
	gTensionLogic.Status.ActProcessedDistance := TensionController[1].Info.ProcessedMaterial - StartingMaterialToProcess;
	ProgressBarProcent :=  (gTensionLogic.Status.ActProcessedDistance / gMainLogic.MotorMode.Production.Parameter.Distance) * 100.0;
	IF gMainLogic.MotorMode.Production.Parameter.Distance = 0.0 OR Status.StateCurrent = 'Stopped' AND Status.StateCurrent = 'Idle' AND THEN
	  ProgressBarProcent := 0.0;
	END_IF;
	IF ProgressBarProcent >= 100.0 OR Status.StateCurrent = 'Stopped' AND Status.StateCurrent = 'Idle' THEN
		StartingMaterialToProcess := TensionController[1].Info.ProcessedMaterial;
	END_IF;

END_ACTION
```

#### actCallBlocks.st
```iecst
ACTION actCallBlocks:
	FOR i := 0 TO INDEX_NR_OF_ZONES DO
		TensionController[i]();
		MpAxisBasicFB[i]();
	END_FOR;
	TensionGroup();
END_ACTION
```

#### actExitTension.st
```iecst
ACTION actExitTension:
	TensionGroup.Enable := FALSE;
	TensionGroup();

	FOR i := 0 TO INDEX_NR_OF_ZONES DO

		TensionController[i].Enable := FALSE;
		TensionController[i]();
		MpAxisBasicFB[i].Enable := FALSE;
		MpAxisBasicFB[i]();

	END_FOR;
END_ACTION
```

#### actSetGlobals.st
```iecst
ACTION actSetGlogals:
	gTensionLogic.Status.ActLeftDancerPos := ActLeftDancerPosScal;
	gTensionLogic.Status.ActRightDancerPos := ActRightDancerPosScal;
	gTensionLogic.Status.LeftWinderDiameter := TensionController[0].Info.DiameterEstimation.EstimatedDiameter;
	gTensionLogic.Status.RightWinderDiameter := TensionController[2].Info.DiameterEstimation.EstimatedDiameter;
	IF TensionController[0].PresetDiameterSet AND TensionController[2].PresetDiameterSet THEN
	  	LeftWinderDiameter := TensionController[0].Info.DiameterEstimation.EstimatedDiameter;
		RightWinderDiameter := TensionController[2].Info.DiameterEstimation.EstimatedDiameter;
	END_IF;

	gTensionLogic.Mode.Manual.Axis1.Parameter.RotarySpeed := MpAxisBasicFB[0].Velocity * 60.0 / 360.0;
	gTensionLogic.Mode.Manual.Axis2.Parameter.LinearSpeed := MpAxisBasicFB[1].Velocity * 60.0 / 1000.0;
	gTensionLogic.Mode.Manual.Axis3.Parameter.RotarySpeed := MpAxisBasicFB[2].Velocity * 60.0 / 360.0;
	gTensionLogic.Mode.Manual.Axis1.Status.IsInMotion := MpAxisBasicFB[0].MoveActive;
	gTensionLogic.Mode.Manual.Axis2.Status.IsInMotion := MpAxisBasicFB[1].MoveActive;
	gTensionLogic.Mode.Manual.Axis3.Status.IsInMotion := MpAxisBasicFB[2].MoveActive;
	gTensionLogic.Status.LineIsHomed := TensionGroup.IsHomed AND gTensionLogic.Status.MasterIsHomed;
	gTensionLogic.Status.LineIsPoweredOn := TensionGroup.PowerOn AND gTensionLogic.Status.MasterIsPowerOn;
	gMainLogic.MotorMode.Production.Status.ActDistance := TensionController[1].Info.ProcessedMaterial;
	gTensionLogic.Status.EnableAxis1 := MpAxisBasicFB[0].Info.DigitalInputsStatus.DriveEnable;
	gTensionLogic.Status.EnableAxis2 := MpAxisBasicFB[1].Info.DigitalInputsStatus.DriveEnable;
	gTensionLogic.Status.EnableAxis3 := MpAxisBasicFB[2].Info.DigitalInputsStatus.DriveEnable;
	gTensionLogic.Status.ProgressBarProcent := ProgressBarProcent;
	gTensionLogic.Status.ErrorExist := TensionController[0].Error OR TensionController[1].Error OR TensionController[2].Error OR TensionGroup.Error;
END_ACTION
```

#### actReadGlobals.st
```iecst
ACTION actReadGlobals:
	TensionController[0].ErrorReset := gMainLogic.MotorMode.Production.Cmd.Reset;
	TensionController[1].ErrorReset := gMainLogic.MotorMode.Production.Cmd.Reset;
	TensionController[2].ErrorReset := gMainLogic.MotorMode.Production.Cmd.Reset;
	TensionGroup.ErrorReset := gMainLogic.MotorMode.Production.Cmd.Reset;

	TensionGroup.Home := gMainLogic.MotorMode.Production.Cmd.Home;

	IF TensionGroup.IsHomed THEN
	  	TensionGroup.Power := gMainLogic.MotorMode.Production.Cmd.PowerOn;
	END_IF;
	TensionGroup.MoveVelocity := gTensionLogic.Status.SetDancers;
	ProgressBarProcent := gTensionLogic.Status.ProgressBarProcent;
//	MpAxisBasicFB[0].ErrorReset := gMainLogic.MotorMode.Manual.Axis1.Cmd.Reset;
//	MpAxisBasicFB[0].Home := gMainLogic.MotorMode.Manual.Axis1.Cmd.Home;
//	IF MpAxisBasicFB[0].IsHomed THEN
//	  	MpAxisBasicFB[0].Power := gMainLogic.MotorMode.Manual.Axis1.Cmd.PowerOn;
//	END_IF;
//	IF MpAxisBasicFB[1].PowerOn THEN
//		MpAxisBasicFB[0].AutoTune := gMainLogic.MotorMode.Manual.Axis1.Cmd.PIDauto;
//		IF gMainLogic.MotorMode.Manual.Axis1.Parameter.Dir THEN
//			MpAxisBasicFB[0].JogPositive := gMainLogic.MotorMode.Manual.Axis1.Cmd.JogAxis;
//		ELSIF NOT(gMainLogic.MotorMode.Manual.Axis1.Parameter.Dir) THEN
//			MpAxisBasicFB[0].JogNegative := gMainLogic.MotorMode.Manual.Axis1.Cmd.JogAxis;
//		END_IF;
//	END_IF;

//	MpAxisBasicFB[1].Home := gMainLogic.MotorMode.Manual.Axis2.Cmd.Home;
//	IF MpAxisBasicFB[1].IsHomed THEN
//		MpAxisBasicFB[1].Power := gMainLogic.MotorMode.Manual.Axis1.Cmd.PowerOn;
//	END_IF;
//	IF MpAxisBasicFB[1].PowerOn THEN
//		MpAxisBasicFB[1].Power := gMainLogic.MotorMode.Manual.Axis2.Cmd.PowerOn;
//		MpAxisBasicFB[1].ErrorReset := gMainLogic.MotorMode.Manual.Axis2.Cmd.Reset;
//		MpAxisBasicFB[1].AutoTune := gMainLogic.MotorMode.Manual.Axis2.Cmd.PIDauto;
//		IF gMainLogic.MotorMode.Manual.Axis2.Parameter.Dir THEN
//			MpAxisBasicFB[1].JogPositive := gMainLogic.MotorMode.Manual.Axis2.Cmd.JogAxis;
//		ELSIF NOT(gMainLogic.MotorMode.Manual.Axis2.Parameter.Dir) THEN
//			MpAxisBasicFB[1].JogNegative := gMainLogic.MotorMode.Manual.Axis2.Cmd.JogAxis;
//		END_IF;
//	END_IF;

//
//	MpAxisBasicFB[2].Home := gMainLogic.MotorMode.Manual.Axis3.Cmd.Home;
//	IF MpAxisBasicFB[2].IsHomed THEN
//		MpAxisBasicFB[2].Power := gMainLogic.MotorMode.Manual.Axis1.Cmd.PowerOn;
//	END_IF;
//	IF MpAxisBasicFB[2].PowerOn THEN
//		MpAxisBasicFB[2].Power := gMainLogic.MotorMode.Manual.Axis3.Cmd.PowerOn;
//		MpAxisBasicFB[2].ErrorReset := gMainLogic.MotorMode.Manual.Axis3.Cmd.Reset;
//		MpAxisBasicFB[2].AutoTune := gMainLogic.MotorMode.Manual.Axis3.Cmd.PIDauto;
//		IF gMainLogic.MotorMode.Manual.Axis3.Parameter.Dir THEN
//			MpAxisBasicFB[2].JogPositive := gMainLogic.MotorMode.Manual.Axis3.Cmd.JogAxis;
//		ELSIF NOT(gMainLogic.MotorMode.Manual.Axis3.Parameter.Dir) THEN
//			MpAxisBasicFB[2].JogNegative := gMainLogic.MotorMode.Manual.Axis3.Cmd.JogAxis;
//		END_IF;
//	END_IF;
//	IF gTensionLogic.Status.SetDancers THEN
	  	SetLeftDancerPos := gMainLogic.MotorMode.Production.Parameter.DancerPos1;
		SetRightDancerPos := gMainLogic.MotorMode.Production.Parameter.DancerPos2;
//		gTensionLogic.Status.SetDancers := FALSE;
//	END_IF;

END_ACTION
```

#### actCatchError.st - not listed in the package file held
```iecst
ACTION actCatchError:
	IF TensionGroup.Error THEN
		step := ERROR;
	END_IF;
END_ACTION
```

#### actExecuteErrorReset.st - not listed in the package file held
```iecst
ACTION actExecuteErrorReset:
	TensionGroup.ErrorReset := TRUE;
	FOR i := 0 TO INDEX_NR_OF_ZONES DO
		TensionController[i].ErrorReset := TRUE;
	END_FOR;
	IF NOT TensionGroup.Error THEN
		FOR i := 0 TO INDEX_NR_OF_ZONES DO
			TensionController[i].ErrorReset := FALSE;
		END_FOR;
		TensionGroup.ErrorReset := FALSE;
		step := INIT;
	END_IF;
END_ACTION
```

#### actExecuteMoveAbsolute.st - not listed in the package file held
```iecst
ACTION actExecuteMoveAbsolute:
	TensionGroup.MoveVelocity := TRUE;
	IF TensionController[1].Info.ProcessedMaterial >= Distance THEN
		TensionGroup.StopLine := TRUE;
		step := WAIT_FOR_COMMAND;
	END_IF;
END_ACTION
```

#### actHandleError.st - not listed in the package file held
```iecst
ACTION actHandleError:
	TensionGroup.MoveVelocity := FALSE;
	TensionGroup.Control := FALSE;
	TensionGroup.Home := FALSE;
	step := ERROR_RESET;
END_ACTION
```

#### actHomeTensionGroup.st - not listed in the package file held
```iecst
ACTION actHomeTensionGroup:
	TensionGroup.Home := TRUE;
	IF TensionGroup.IsHomed THEN
		TensionGroup.Home := FALSE;
		step := POWER;
	END_IF;
END_ACTION
```

#### actInitTensionGroup.st - not listed in the package file held
```iecst
ACTION actInitTencionGroup:
	TensionGroup.Enable := TRUE;
	TensionGroup.Home := FALSE;
	TensionGroup.Power := FALSE;
	step := HOME;
END_ACTION
```

#### actPowerOnTensionGroup.st - not listed in the package file held
```iecst
ACTION actPowerOnTensionGroup:
	TensionGroup.Power := TRUE;
	IF TensionGroup.PowerOn THEN
		step := WAIT_FOR_COMMAND;
	END_IF;
END_ACTION
```

#### actWaitForCommand.st - not listed in the package file held
```iecst
ACTION actWaitForCommand:
	TensionGroup.MoveVelocity := TRUE;
END_ACTION
```

#### ReadGlobals.st - not listed in the package file held
```iecst
ACTION ReadGlobals:

END_ACTION
```

#### SetGlobals.st - not listed in the package file held
```iecst
ACTION SetGlogals:
	gTensionLogic.Status.ActLeftDancerPos := ActLeftDancerPosScal;
	gTensionLogic.Status.ActRightDancerPos := ActRightDancerPosScal;
	gTensionLogic.Status.LeftWinderDiameter := TensionController[0].Info.DiameterEstimation.EstimatedDiameter;
	gTensionLogic.Status.RightWinderDiameter := TensionController[2].Info.DiameterEstimation.EstimatedDiameter;
	gTensionLogic.Mode.Manual.Axis1.Parameter.RotarySpeed := MpAxisBasicFB[0].Velocity;
	gTensionLogic.Mode.Manual.Axis2.Parameter.LinearSpeed := MpAxisBasicFB[1].Velocity;
	gTensionLogic.Mode.Manual.Axis3.Parameter.RotarySpeed := MpAxisBasicFB[2].Velocity;
END_ACTION
```

#### InitAxis.st - not listed in the package file held
```iecst
ACTION actInitAxes:
	FOR i := 0 TO 2 DO
		Axis[i].AxisBasic.Enable := TRUE;
		Axis[i].AxisPar.Deafult.Acceleration := 20.0;
		Axis[i].AxisPar.Deafult.Deceleration := 20.0;
		Axis[i].AxisPar.Deafult.Position := 10.0;
		Axis[i].AxisPar.Deafult.Distance := 20;
		Axis[i].AxisPar.Deafult.Homing.Mode := mcHOMING_DIRECT;
		Axis[i].AxisPar.Deafult.Homing.Position := 0;
		Tension.TensionController[i].Control := TRUE;
		Tension.TensionGroup.Control := TRUE;
	END_FOR;
END_ACTION
```

#### PrepForWork.st - not listed in the package file held
```iecst
ACTION actPrepForWork:
	FOR i := 0 TO 2 DO
		IF Tension.TensionController[i].Error THEN
			Control.Step[i] := ERROR;
		END_IF;
		CASE Control.Step[i] OF
			COMMUNICATION:
				IF Axis[i].AxisBasic.Info.CommunicationReady AND Axis[i].AxisBasic.Info.ReadyToPowerOn AND Tension.TensionController[i].ControlBusy AND Tension.TensionGroup.ControlBusy THEN
	  				Control.Step[i] := HOME;
				END_IF;
			HOME:
				Tension.TensionGroup.Home := TRUE;
				IF Tension.TensionGroup.IsHomed THEN
					Tension.TensionGroup.Home := FALSE;
					Control.Step[i] := POWER;
				END_IF;
			POWER:
				Tension.TensionGroup.Power := TRUE;
				IF Tension.TensionGroup.PowerOn THEN
	  				Control.Step[i] := READY_FOR_USE;
				END_IF;
			ERROR:
				Tension.TensionGroup.Power := FALSE;
				Control.Step[i] := ERROR_RESET;
			ERROR_RESET:
				Tension.TensionGroup.ErrorReset := TRUE;
				IF Tension.TensionGroup.Error THEN
					Tension.TensionGroup.ErrorReset := FALSE;
					Control.Step[i] := COMMUNICATION;
				END_IF;
		END_CASE;
	END_FOR;
END_ACTION
```

### Program Logical/Control/Tension/TensionConfig (IEC)

#### TensionVarConfig.var - Local variables
```iecst
VAR
	TensionConfigType : ARRAY[0..2] OF MpTensionControllerConfigType;
	TensionConfig : ARRAY[0..2] OF MpTensionControllerConfig;
	gAxisString1 : STRING[32] := 'gAxis_1';
	SetLeftDancerPos : STRING[255] := '::Tension:SetLeftDancerPos';
	ActLeftDancerPosScal : STRING[255] := '::Tension:ActLeftDancerPosScal';
	gAxisString3 : STRING[32] := 'gAxis_3';
	SetRightDancerPos : STRING[255] := '::Tension:SetRightDancerPos';
	ActRightDancerPosScal : STRING[255] := '::Tension:ActRightDancerPosScal';
	gAxisString2 : STRING[32] := 'gAxis_2';
	StepPID2 : ConfigPID2 := ACTIV_PID2;
	StepPID1 : ConfigPID1 := ACTIV_PID1;
END_VAR
```

#### TensionTypConfig.typ - Local data types
```iecst
TYPE
	ConfigPID2 :
		(
		ACTIV_PID2,
		START_PID2,
		WAIT_PID2,
		FINISH_PID2
		);
	ConfigPID1 :
		(
		ACTIV_PID1,
		START_PID1,
		WAIT_PID1,
		FINISH_PID1
		);
END_TYPE
```

#### TensionGroupConfig.st - Init, cyclic, exit code
```iecst
PROGRAM _INIT
	actInitTensionConfig;
END_PROGRAM

PROGRAM _CYCLIC
	actCallTensionConfig;

//	TensionConfig[0].Load := TRUE;
//	TensionConfig[1].Load := TRUE;
//	TensionConfig[2].Load := TRUE;
	actConfigAxis1;
	actConfigAxis3;

//	TensionConfig[0].Save := TRUE;
//	TensionConfig[1].Save := TRUE;
//	TensionConfig[2].Save := TRUE;

END_PROGRAM

PROGRAM _EXIT

	actExitTensionConfig;

END_PROGRAM
```

#### actConfigAxis1.st
```iecst
ACTION actConfigAxis1:

	CASE StepPID1 OF

		ACTIV_PID1:
			IF TensionConfig[0].Active THEN
				StepPID1 := START_PID1;
			END_IF;

		START_PID1:
			TensionConfig[0].Load := TRUE;
			IF TensionConfig[0].CommandDone THEN
				TensionConfig[0].Load := FALSE;
				gHMI.Recipe.CurrentRecipe.Dencer1PID.P := TensionConfigType[0].Controller.PIDParameters.OperatingPoint1.ProportionalGain;
				gHMI.Recipe.CurrentRecipe.Dencer1PID.I := TensionConfigType[0].Controller.PIDParameters.OperatingPoint1.IntegrationTime;
				StepPID1 := WAIT_PID1;
			END_IF;

		WAIT_PID1:
			IF gHMI.Recipe.Load THEN
				StepPID1 := FINISH_PID1;
			END_IF;

		FINISH_PID1:
			TensionConfigType[0].Controller.PIDParameters.OperatingPoint1.ProportionalGain := gHMI.Recipe.CurrentRecipe.Dencer1PID.P;
			TensionConfigType[0].Controller.PIDParameters.OperatingPoint1.IntegrationTime := gHMI.Recipe.CurrentRecipe.Dencer1PID.I;
			TensionConfig[0].Save := TRUE;
			IF TensionConfig[0].CommandDone THEN
				TensionConfig[0].Save := FALSE;
				StepPID1 := WAIT_PID1;
			END_IF;

	END_CASE;
END_ACTION
```

#### actConfigAxis2.st
```iecst
ACTION actConfigAxis2:

END_ACTION
```

#### actConfigAxis3.st
```iecst
ACTION actConfigAxis3:

	CASE StepPID2 OF

		ACTIV_PID2:
			IF TensionConfig[2].Active THEN
				StepPID2 := START_PID2;

			END_IF;

		START_PID2:
			TensionConfig[2].Load := TRUE;
			IF TensionConfig[2].CommandDone THEN
				TensionConfig[2].Load := FALSE;
				gHMI.Recipe.CurrentRecipe.Dencer1PID.P := TensionConfigType[2].Controller.PIDParameters.OperatingPoint1.ProportionalGain;
				gHMI.Recipe.CurrentRecipe.Dencer1PID.I := TensionConfigType[2].Controller.PIDParameters.OperatingPoint1.IntegrationTime;
				StepPID2 := WAIT_PID2;
			END_IF;

		WAIT_PID2:
			IF gHMI.Recipe.Load THEN
				StepPID2 := FINISH_PID2;
			END_IF;

		FINISH_PID2:
			TensionConfigType[2].Controller.PIDParameters.OperatingPoint1.ProportionalGain := gHMI.Recipe.CurrentRecipe.Dencer1PID.P;
			TensionConfigType[2].Controller.PIDParameters.OperatingPoint1.IntegrationTime := gHMI.Recipe.CurrentRecipe.Dencer1PID.I;
			TensionConfig[2].Save := TRUE;
			IF TensionConfig[2].CommandDone THEN
				TensionConfig[2].Save := FALSE;
				StepPID2 := WAIT_PID2;
			END_IF;

	END_CASE;
END_ACTION
```

#### actInitTensionConfig.st
```iecst
ACTION actInitTensionConfig:
	// MpLink
	TensionConfig[0].MpLink := ADR(gTensionCtrl_Unwinder);
	TensionConfig[1].MpLink := ADR(gTensionCtrl_Master);
	TensionConfig[2].MpLink := ADR(gTensionCtrl_Rewinder);

	TensionConfig[0].Enable := TRUE;
	TensionConfig[1].Enable := TRUE;
	TensionConfig[2].Enable := TRUE;

END_ACTION
```

#### actCallTensionConfig.st
```iecst
ACTION actCallTensionConfig:

	TensionConfig[0].Configuration := ADR( TensionConfigType[0]);
	TensionConfig[0]();

	TensionConfig[1].Configuration := ADR( TensionConfigType[1]);
	TensionConfig[1]();

	TensionConfig[2].Configuration := ADR( TensionConfigType[2]);
	TensionConfig[2]();
END_ACTION
```

#### actExitTensionConfig.st
```iecst
ACTION actExitTensionConfig:
	TensionConfig[0].Enable := FALSE;
	TensionConfig[0]();

	TensionConfig[1].Enable := FALSE;
	TensionConfig[1]();

	TensionConfig[2].Enable := FALSE;
	TensionConfig[2]();
END_ACTION
```

#### actExitConfig.st - not listed in the package file held
```iecst
ACTION actExitConfig:
	// Enable
	TensionConfig[0].Enable := FALSE;
	TensionConfig[0]();

	TensionConfig[1].Enable := FALSE;
	TensionConfig[1]();

	TensionConfig[2].Enable := FALSE;
	TensionConfig[2]();
END_ACTION
```

#### actInitAxisLeft.st - not listed in the package file held
```iecst
ACTION actInitAxisLeft:
	// Pierwszy Axis
	TensionConfigType[0].MotionSystem.AxisReference := gAxisString1;
	TensionConfigType[0].MotionSystem.AxisVelocityProfile.Acceleration := 0.1;
	TensionConfigType[0].MotionSystem.AxisVelocityProfile.Deceleration := 0.5;
	TensionConfigType[0].MotionSystem.AxisVelocityProfile.StopDeceleration := 2.0;
	TensionConfigType[0].MotionSystem.AxisVelocityProfile.JerkTime := 0.0;

	TensionConfigType[0].Utilization.Winder.Width := 1000.0;
	TensionConfigType[0].Utilization.Winder.MinimumDiameter := 30.0;
	TensionConfigType[0].Utilization.Winder.MaximumDiameter := 80.0;
	TensionConfigType[0].Utilization.Winder.Winding := mpTENSION_WINDING_FROM_TOP;
	TensionConfigType[0].Utilization.DiameterEstimation.EstimationWindow := mpTENSION_EST_MODE_POSITION;

	TensionConfigType[0].Controller.Type := mpTENSION_CONTROL_DANCER;
	TensionConfigType[0].Controller.Mode := mpTENSION_CONTROL_CLOSED_LOOP;
	TensionConfigType[0].Controller.PIDParameters.OperatingPoint1.ProportionalGain := 5.0;
	TensionConfigType[0].Controller.PIDParameters.OperatingPoint1.IntegrationTime := 0.0;
	TensionConfigType[0].Controller.PIDParameters.OperatingPoint1.DerivativeTime := 0.0;
	TensionConfigType[0].Controller.PIDParameters.OperatingPoint1.FilterTime := 0.0;
	TensionConfigType[0].Controller.MaximumVelocityCorrection := 10.0;
	TensionConfigType[0].Controller.ToleranceBand.Lower := 4.0;
	TensionConfigType[0].Controller.ToleranceBand.Upper := 4.0;
	TensionConfigType[0].Controller.Initialization.MaximumLineVelocityCorrection := 10.0;
	TensionConfigType[0].Controller.Initialization.SettlingTime := 1.0;
	TensionConfigType[0].Controller.Initialization.TimeOut := 30.0;

	TensionConfigType[0].Material.Length := 0.4;
	TensionConfigType[0].Material.Thickness := 80.0;
	TensionConfigType[0].Material.Width := 48.0;
	TensionConfigType[0].Material.YoungsModulus := 400000000.0;
	TensionConfigType[0].Material.TensionLimit := 300.0;
	TensionConfigType[0].InputSignals.SetDancerPosition := SetLeftDancerPos;
	TensionConfigType[0].InputSignals.ActualDancerPosition := ActLeftDancerPosScal;

END_ACTION
```

#### actInitAxisMid.st - not listed in the package file held
```iecst
ACTION actInitAxisMid:
	// Drugi Axis
	TensionConfigType[1].MotionSystem.AxisReference := gAxisString2;
	TensionConfigType[1].MotionSystem.AxisVelocityProfile.Acceleration := 0.1;
	TensionConfigType[1].MotionSystem.AxisVelocityProfile.Deceleration := 0.5;
	TensionConfigType[1].MotionSystem.AxisVelocityProfile.StopDeceleration := 2.0;
	TensionConfigType[1].MotionSystem.AxisVelocityProfile.JerkTime := 0.0;
END_ACTION
```

#### actInitAxisRight.st - not listed in the package file held
```iecst
ACTION actInitAxisRight:
	// Trzeci Axis
	TensionConfigType[2].MotionSystem.AxisReference := gAxisString3;
	TensionConfigType[2].MotionSystem.AxisVelocityProfile.Acceleration := 0.1;
	TensionConfigType[2].MotionSystem.AxisVelocityProfile.Deceleration := 0.5;
	TensionConfigType[2].MotionSystem.AxisVelocityProfile.StopDeceleration := 2.0;
	TensionConfigType[2].MotionSystem.AxisVelocityProfile.JerkTime := 0.0;

	TensionConfigType[2].Utilization.Winder.Width := 1000.0;
	TensionConfigType[2].Utilization.Winder.MinimumDiameter := 30.0;
	TensionConfigType[2].Utilization.Winder.MaximumDiameter := 80.0;
	TensionConfigType[2].Utilization.Winder.Winding := mpTENSION_WINDING_FROM_TOP;
	TensionConfigType[2].Utilization.DiameterEstimation.EstimationWindow := mpTENSION_EST_MODE_POSITION;

	TensionConfigType[2].Controller.Type := mpTENSION_CONTROL_DANCER;
	TensionConfigType[2].Controller.Mode := mpTENSION_CONTROL_CLOSED_LOOP;
	TensionConfigType[2].Controller.PIDParameters.OperatingPoint1.ProportionalGain := 5.0;
	TensionConfigType[2].Controller.PIDParameters.OperatingPoint1.IntegrationTime := 0.0;
	TensionConfigType[2].Controller.PIDParameters.OperatingPoint1.DerivativeTime := 0.0;
	TensionConfigType[2].Controller.PIDParameters.OperatingPoint1.FilterTime := 0.0;
	TensionConfigType[2].Controller.MaximumVelocityCorrection := 10.0;
	TensionConfigType[2].Controller.ToleranceBand.Lower := 4.0;
	TensionConfigType[2].Controller.ToleranceBand.Upper := 4.0;
	TensionConfigType[2].Controller.Initialization.MaximumLineVelocityCorrection := 10.0;
	TensionConfigType[2].Controller.Initialization.SettlingTime := 1.0;
	TensionConfigType[2].Controller.Initialization.TimeOut := 30.0;

	TensionConfigType[2].Material.Length := 0.4;
	TensionConfigType[2].Material.Thickness := 80.0;
	TensionConfigType[2].Material.Width := 48.0;
	TensionConfigType[2].Material.YoungsModulus := 400000000.0;
	TensionConfigType[2].Material.TensionLimit := 300.0;
	TensionConfigType[2].InputSignals.SetDancerPosition := SetRightDancerPos;
	TensionConfigType[2].InputSignals.ActualDancerPosition := ActRightDancerPosScal;

END_ACTION
```

#### actInitEnable.st - not listed in the package file held
```iecst
ACTION actInitEnable:
	//InitEnable
	TensionConfig[0].Enable := TRUE;
	TensionConfig[1].Enable := TRUE;
	TensionConfig[2].Enable := TRUE;

END_ACTION
```

#### actMainLoop.st - not listed in the package file held
```iecst
ACTION actMainLoop:
	// Cyclic
	TensionConfig[0]();
	TensionConfig[1]();
	TensionConfig[2]();

END_ACTION
```

#### actMplink.st - not listed in the package file held
```iecst
ACTION actMplink:
	// MpLink
	TensionConfig[0].MpLink := ADR(gTensionCtrl_Unwinder);
	TensionConfig[1].MpLink := ADR(gTensionCtrl_Master);
	TensionConfig[2].MpLink := ADR(gTensionCtrl_Rewinder);
END_ACTION
```

### gTensiontype.typ
```iecst
TYPE
	gTensionLogicType : 	STRUCT
		Mode : WorkModeType;
		Cmd : CommandTensionType;
		Parameter : ParameterTensionType;
		Status : StatusTensionType;
	END_STRUCT;
	CommandTensionType : 	STRUCT
		SetRightDancerPos : REAL; (*sets position of right dancer in mm*)
		SetLeftDancerPos : REAL; (*sets position of left dancer in mm*)
	END_STRUCT;
	ParameterTensionType : 	STRUCT
		GroupLineVelocity : REAL; (*in m/min*)
	END_STRUCT;
	StatusTensionType : 	STRUCT
		ActRightDancerPos : REAL; (*actual right dancer position in mm*)
		ActLeftDancerPos : REAL; (*actual left dancer position in mmm*)
		LeftWinderDiameter : REAL; (*diameter on left winder*)
		RightWinderDiameter : REAL; (*diameter on right winder*)
		LineIsInMove : BOOL; (*checks if line is moving*)
		LineIsHomed : BOOL; (*checks if line is homed*)
		LineIsPoweredOn : BOOL; (*checks if line is powered on*)
		MasterIsPowerOn : BOOL; (*inside variable to communicate beatween programs*)
		MasterIsHomed : BOOL; (*inside variable to communicate beatween programs*)
		EnableAxis1 : BOOL; (*chacks if left axis is enabled*)
		EnableAxis2 : BOOL; (*chacks if middle axis is enabled*)
		EnableAxis3 : BOOL; (*chacks if right axis is enabled*)
		ProgressBarProcent : REAL; (*procent for progress bar*)
		ErrorExist : BOOL;
		ActProcessedDistance : REAL; (*proceset distance from executed state*)
		SetDancers : BOOL; (*force dancers to set position on riseing edge*)
		MoveDone : BOOL;
	END_STRUCT;
	WorkModeType : 	STRUCT
		Production : ProdLogicType;
		Manual : ManAxisSelectType;
	END_STRUCT;
	ProdLogicType : 	STRUCT
		a : BOOL;
	END_STRUCT;
	ManAxisSelectType : 	STRUCT
		Axis1 : Axis1LogType;
		Axis2 : Axis2LogType;
		Axis3 : Axis3LogType;
	END_STRUCT;
	Axis1LogType : 	STRUCT
		Parameter : Axis1ParaType;
		Status : Axis1StatType;
	END_STRUCT;
	Axis2LogType : 	STRUCT
		Parameter : Axis2ParaType;
		Status : Axis2StatType;
	END_STRUCT;
	Axis3LogType : 	STRUCT
		Parameter : Axis3ParaType;
		Status : Axis3StatType;
	END_STRUCT;
	Axis1ParaType : 	STRUCT
		RotarySpeed : REAL; (*rpm*)
		Axis1DancerPara : Axis1ParaDancerPID;
		Axis1PID : Axis1ParaPID;
	END_STRUCT;
	Axis1ParaDancerPID : 	STRUCT
		P : REAL;
		I : REAL;
		D : REAL;
	END_STRUCT;
	Axis1ParaPID : 	STRUCT
		P : REAL;
		I : REAL;
		D : REAL;
	END_STRUCT;
	Axis1StatType : 	STRUCT
		IsInMotion : BOOL; (*checks if axis is in motion*)
	END_STRUCT;
	Axis2ParaType : 	STRUCT
		LinearSpeed : REAL; (*m/min*)
		Axis2PID : Axis2ParaPID;
	END_STRUCT;
	Axis2ParaPID : 	STRUCT
		P : REAL;
		I : REAL;
		D : REAL;
	END_STRUCT;
	Axis2StatType : 	STRUCT
		IsInMotion : BOOL; (*checks if axis is in motion*)
	END_STRUCT;
	Axis3ParaType : 	STRUCT
		RotarySpeed : REAL; (*in rpm*)
		Axis3DancerPara : Axis3ParaDancerPID;
		Axis3PID : Axis3ParaPID;
	END_STRUCT;
	Axis3ParaDancerPID : 	STRUCT
		P : REAL;
		I : REAL;
		D : REAL;
	END_STRUCT;
	Axis3ParaPID : 	STRUCT
		P : REAL;
		I : REAL;
		D : REAL;
	END_STRUCT;
	Axis3StatType : 	STRUCT
		IsInMotion : BOOL; (*checks if axis is in motion*)
	END_STRUCT;
END_TYPE
```

### gTensionVar.var
```iecst
VAR
	gTensionLogic : gTensionLogicType;
END_VAR
```

### Program Logical/Control/Tension/VAxis (IEC)

#### VAxis.st - Init, cyclic, exit code
```iecst
PROGRAM _INIT
	MpAxisBasicMaster.MpLink := ADR(gAxisMaster);
	MpAxisBasicMaster.Enable := TRUE;
	MpAxisBasicMasterPar.Position := 100.0;
	MpAxisBasicMasterPar.Distance := 1000.0;
	MpAxisBasicMasterPar.Velocity := 500.0;
	MpAxisBasicMasterPar.Acceleration := 100.0;
	MpAxisBasicMasterPar.Deceleration := 100.0;
	MpAxisBasicMasterPar.Jog.Velocity := 500.0;
	MpAxisBasicMasterPar.Jog.Acceleration := 10.0;
	MpAxisBasicMasterPar.Jog.Deceleration := 10.0;
	MpAxisBasicMaster.Parameters := ADR(MpAxisBasicMasterPar);
	PowerStep := POWER_INIT;
END_PROGRAM

PROGRAM _CYCLIC

	MpAxisBasicMaster.Power := gMainLogic.MotorMode.Production.Cmd.PowerOn;
	MpAxisBasicMaster.Home := gMainLogic.MotorMode.Production.Cmd.Home;
	MpAxisBasicMaster.ErrorReset := gMainLogic.MotorMode.Production.Cmd.Reset;
	MpAxisBasicMaster.MoveAdditive := gMainLogic.MotorMode.Production.Cmd.StartWinding;
	MpAxisBasicMaster.MoveVelocity := gMainLogic.MotorMode.Manual.JogWithTenReg;
	MpAxisBasicMaster.Stop := gMainLogic.MotorMode.Production.Cmd.EmergencyStop;

	MpAxisBasicMasterPar.Velocity := gMainLogic.MotorMode.Production.Parameter.Velocity * 1000.0/ 60.0;
	MpAxisBasicMasterPar.Distance := gMainLogic.MotorMode.Production.Parameter.Distance * 1000.0;

	LineVelocityInMeters := MpAxisBasicMaster.Velocity * 60.0 / 1000.0;

	gTensionLogic.Parameter.GroupLineVelocity := LineVelocityInMeters;
	gTensionLogic.Status.MasterIsHomed := MpAxisBasicMaster.IsHomed;
	gTensionLogic.Status.MasterIsPowerOn := MpAxisBasicMaster.PowerOn;
	gMainLogic.MotorMode.Production.Status.ActVelocity := LineVelocityInMeters;
	gTensionLogic.Status.ErrorExist := MpAxisBasicMaster.Error;
	gTensionLogic.Status.MoveDone := MpAxisBasicMaster.MoveDone;
	MpAxisBasicMaster();

END_PROGRAM

PROGRAM _EXIT
	MpAxisBasicMaster.Enable := FALSE;
	MpAxisBasicMaster();
END_PROGRAM
```

#### VAxisType.typ - Local data types
```iecst
TYPE
	PowerState :
		(
		POWER_INIT,
		POWER_REQUEST_ON,
		POWER_CHECK_ON,
		POWER_DONE
		);
END_TYPE
```

#### VAxisVar.var - Local variables
```iecst
VAR
	PowerStep : PowerState;
	MpAxisBasicMasterPar : MpAxisBasicParType;
	MpAxisBasicMaster : MpAxisBasic;
	LineVelocityInMeters : REAL;
	PrevVelocity : REAL;
	PrevDistance : REAL;
	UpdateEdge : BOOL;
	UpdateTrigger : BOOL;
END_VAR
```

### gTensionLogicalType.typ - not listed in the package file held
```iecst
TYPE
	(*Enumeration for the tension control state machine, renamed for clarity from TESTstate*)
	TensionStateEnum :
		(
		TNS_INIT,
		TNS_POWER,
		TNS_ERROR,
		TNS_ERROR_RESET,
		TNS_HOME,
		TNS_WAIT_FOR_COMMAND,
		TNS_MOVE_ABSOLUTE
	);

	(*Structure to group the Process Variable (PV) name configurations*)
	TensionPV_ConfigType : STRUCT
		SetLeftDancerPos : STRING[255];
		ActLeftDancerPosScal : STRING[255];
		SetRightDancerPos : STRING[255];
		ActRightDancerPosScal : STRING[255];
	END_STRUCT;

	(*Structure for all configuration and parameters*)
	TensionParType : STRUCT
		ConfigType : ARRAY[0..2] OF MpTensionControllerConfigType;
		Config : ARRAY[0..2] OF MpTensionControllerConfig;
		AxisNames : ARRAY[0..2] OF STRING[32];
		PV_Names : TensionPV_ConfigType;
		SetLeftDancerPos : REAL;
		SetRightDancerPos : REAL;
		GroupLineVelocity : REAL;
	END_STRUCT;

	(*Structure for all status feedback and actual process values*)
	TensionStatusType : STRUCT
		RightWinderDiameter : REAL;
		LeftWinderDiameter : REAL;
		ActLeftDancerPos : INT;
		ActLeftDancerPosScal : REAL;
		ActRightDancerPos : INT;
		ActRightDancerPosScal : REAL;
	END_STRUCT;

	(*Structure for internal variables and function block instances*)
	TensionInternalType : STRUCT
		Controller : ARRAY[0..2] OF MpTensionController;
		Group : MpTensionGroup;
		MvAbsActive : BOOL;
		LoopIndex : USINT;
	END_STRUCT;

	(*Main global structure for the entire tension control program*)
	gTensionLogicType : STRUCT
		State : TensionStateEnum;
		Par : TensionParType;
		Status : TensionStatusType;
		Internal : TensionInternalType;
	END_STRUCT;

END_TYPE
```

### Constants.var - not listed in the package file held
```iecst
VAR CONSTANT
	NR_OF_ZONES : USINT := 3;
	INDEX_NR_OF_ZONES : USINT := NR_OF_ZONES-1;
END_VAR
```

### Variables.var - not listed in the package file held
```iecst
VAR
	gLineSpeed : REAL;
END_VAR
```

### Program Logical/Control/Tension/Dencers (IEC)

#### Dencers.st - Init, cyclic, exit code
```iecst
PROGRAM _INIT
	FOR i :=0 TO 1 DO
		DancerController[i].Enable := 0;
		DancerController[i].Configuration.Geometry.WinderWidth := 95.0;
		DancerController[i].Configuration.Geometry.MaterialThickness := 18.0;
		DancerController[i].Configuration.Geometry.MaxDiameter := 80.0;
		DancerController[i].Configuration.Geometry.MinDiameter := 30.0;
		DancerController[i].Configuration.Geometry.MinInertia := 0.00000001;
		DancerController[i].Configuration.Geometry.TestDiameter := 50.0;
		DancerController[i].Configuration.Geometry.TestInertia := 0.000001;
		DancerController[i].Configuration.Axis.LineUnits := 135617;
		DancerController[i].Configuration.Axis.WinderUnits := 360000; (* 1 winder (unit) == 0.001° *)
		DancerController[i].Configuration.Axis.RevMotor := 1;
		DancerController[i].Configuration.Axis.GearRatio := 3.0; (* gear ratio = 1 *)
		DancerController[i].Configuration.Axis.WinderType := mtWND_UNWIND; (* unwinding system *)
		DancerController[i].Parameters.PIDParameters.Gain := 2.0;
		DancerController[i].Parameters.PIDParameters.IntegrationTime := 1.0;
		DancerController[i].Parameters.PIDParameters.DerivativeTime := 0.0;
		DancerController[i].Parameters.PIDParameters.FilterTime := 0.0;
		DancerController[i].Parameters.MaxLineVelocityCorrection := 1000.0; (* == 1 m/s *)
		DancerController[i].Parameters.MaxControlError := 0.0; (* material break detection off *)

		SetDancerPosition := 10000.0;
		ActDiameter := DancerController[i].Configuration.Geometry.MaxDiameter;
	END_FOR;

END_PROGRAM
PROGRAM _CYCLIC
//	ActDencerPositionMilimeters1 := (ActDancerPosition1 *(1/DancerController[0].Configuration.Axis.LineUnits))/1000;
//	ActDencerPositionMilimeters2 := (ActDancerPosition2 *(1/DancerController[1].Configuration.Axis.LineUnits))/1000;
	FOR i := 0 TO 1 DO
		DancerController[i].Update := TRUE;
		DancerController[i].SetDancerPosition := SetDancerPosition;
		//DancerController[0].ActDancerPosition := ActDencerPositionMilimeters1;
		//DancerController[1].ActDancerPosition := ActDencerPositionMilimeters2;
		DancerController[0].ActDancerPosition := ActDancerPosition1;
		DancerController[1].ActDancerPosition := ActDancerPosition2;
		DancerController[i].ActDiameter := ActDiameter;
		DancerController[i]();
		VelocityCorrection := (DancerController[0].VelocityCorrection + DancerController[1].VelocityCorrection)/2;
		IF DancerController[i].UpdateDone THEN
			DancerController[i].Update := FALSE;
		END_IF;
	END_FOR;
END_PROGRAM

PROGRAM _EXIT
	(* Insert code here *)

END_PROGRAM
```

#### DencersVar.var - Local variables
```iecst
VAR
	DancerController : ARRAY[0..1] OF MTWinderDancerController; (*tension controller*)
	SetDancerPosition : REAL; (*set material tension*)
	ActDancerPosition2 : INT;
	ActDancerPosition1 : INT;
	i : INT;
	ActDiameter : REAL;
	VelocityCorrection : REAL;
	ActDencerPositionMilimeters1 : REAL;
	ActDencerPositionMilimeters2 : REAL;
END_VAR
```

### gAxisType.typ - not listed in the package file held
```iecst
TYPE
	ControlTypeTension : 	STRUCT
		Step : ARRAY[0..2]OF InitState;
		WorkStep : ARRAY[0..2]OF WorkState;
	END_STRUCT;
	WorkState :
		(
		TEST_COMMAND,
		WAIT_FOR_WORK_COMMAND
		);
	InitState :
		(
		COMMUNICATION,
		POWER,
		HOME,
		ERROR,
		READY_FOR_USE,
		ERROR_RESET,
		WAIT_FOR_COMMAND
		);
END_TYPE
```

### gAxisVar.var - not listed in the package file held
```iecst
VAR
	TestAll : BOOL;
	Control : ControlTypeTension;
END_VAR
```

### lAxisType.typ
```iecst
TYPE
	AxisParType : 	STRUCT
		Deafult : MpAxisBasicParType;
	END_STRUCT;
	AxisType : 	STRUCT
		AxisBasic : MpAxisBasic;
		AxisPar : AxisParType;
	END_STRUCT;
END_TYPE
```

### lAxisVar.var
```iecst
VAR
	Axis : ARRAY[0..2] OF AxisType;
END_VAR
```

### Program Logical/Control/Axis/Axis1/Axis1 (IEC)

#### Axis1.st - Init, cyclic, exit code
```iecst
PROGRAM _INIT

END_PROGRAM

PROGRAM _CYCLIC

END_PROGRAM

PROGRAM _EXIT

END_PROGRAM
```

#### Axis1Var.var - Local variables
```iecst
VAR
	Axis1 : Axis;
END_VAR
```

### Program Logical/Control/Axis/Axis2/Axis2 (IEC)

#### Axis2Var.var - Local variables
```iecst
VAR
	Axis2 : Axis;
END_VAR
```

### Program Logical/Control/Axis/Axis3/Axis3 (IEC)

#### Axis3Var.var - Local variables
```iecst
VAR
	Axis3 : Axis;
END_VAR
```

### Program Logical/Control/Axis/Axes (IEC)

#### Axes.st - Init, cyclic, exit code
```iecst
PROGRAM _INIT

END_PROGRAM

PROGRAM _CYCLIC

END_PROGRAM

PROGRAM _EXIT

END_PROGRAM
```

#### AxesVar.var
```iecst
VAR
	Control : ControlType;
END_VAR
```

#### actBlocksInit.st - not listed in the package file held
```iecst
ACTION actBlocksInit:
	FOR i := 0 TO 2 DO
		Axis[i].AxisBasic.Parameters := ADR(Axis[i].AxisPar.Deafult);
		Axis[i].AxisBasic();
	END_FOR;
	Axis[0].AxisBasic.MpLink := ADR(gAxis_1);
	Axis[1].AxisBasic.MpLink := ADR(gAxis_2);
	Axis[2].AxisBasic.MpLink := ADR(gAxis_3);

END_ACTION
```

#### InitAxis.st - not listed in the package file held
```iecst
ACTION actInitAxes:
	FOR i := 0 TO 2 DO
		Axis[i].AxisBasic.Enable := TRUE;
		Axis[i].AxisPar.Deafult.Acceleration := 20.0;
		Axis[i].AxisPar.Deafult.Deceleration := 20.0;
		Axis[i].AxisPar.Deafult.Position := 10.0;
		Axis[i].AxisPar.Deafult.Distance := 20;
		Axis[i].AxisPar.Deafult.Homing.Mode := mcHOMING_DIRECT;
		Axis[i].AxisPar.Deafult.Homing.Position := 0;
	END_FOR;
END_ACTION
```

#### PrepForWork.st - not listed in the package file held
```iecst
ACTION actPrepForWork:
	FOR i := 0 TO 2 DO
		IF Axis[i].AxisBasic.Error THEN
			Control.Step[i] := ERROR;
		END_IF;
		CASE Control.Step[i] OF
			COMMUNICATION:
				IF Axis[i].AxisBasic.Info.CommunicationReady AND Axis[i].AxisBasic.Info.ReadyToPowerOn THEN
	  				Control.Step[i] := HOME;
				END_IF;
			HOME:
				Axis[i].AxisBasic.Home := TRUE;
				IF Axis[i].AxisBasic.IsHomed THEN
					Axis[i].AxisBasic.Home := FALSE;
					Control.Step[i] := POWER;
				END_IF;
			POWER:
				Axis[i].AxisBasic.Power := TRUE;
				IF Axis[i].AxisBasic.PowerOn THEN
	  				Control.Step[i] := READY_FOR_USE;
				END_IF;
			ERROR:
				Axis[i].AxisBasic.Power := FALSE;
				Control.Step[i] := ERROR_RESET;
			ERROR_RESET:
				Axis[i].AxisBasic.ErrorReset := TRUE;
				IF Axis[i].AxisBasic.Error THEN
					Axis[i].AxisBasic.ErrorReset := FALSE;
					Control.Step[i] := COMMUNICATION;
				END_IF;
		END_CASE;
	END_FOR;
END_ACTION
```

### Program Logical/Control/SynMotion/SynMotion (IEC)

#### SynMotion.st - Init, cyclic, exit code
```iecst
PROGRAM _INIT

END_PROGRAM

PROGRAM _CYCLIC

END_PROGRAM

PROGRAM _EXIT

END_PROGRAM
```

### gProgramsType.typ
```iecst
TYPE
	StepEnum :
		(
		STEP_STOPPED, (*STATE_STOPPED*)
		STEP_RESETTING, (*STATE_RESETTING*)
		STEP_IDLE, (*STATE_IDLE*)
		STEP_STARTING, (*STATE_STARTING*)
		STEP_EXECUTE, (*STATE_EXECUTE*)
		STEP_COMPLETING, (*STATE_COMPLETING*)
		STEP_COMPLETE, (*STATE_COMPLETE*)
		STEP_STOPPING, (*STATE_STOPPING*)
		STEP_ABORTING, (*STATE_ABORTING*)
		STEP_ABORTED, (*STATE_ABORTED*)
		STEP_CLEARING (*STATE_CLEARING*)
	);
	ControlTypeMain : 	STRUCT
		Cmd : ControlCmdType;
		Parameter : ControlParType;
		Status : ControlStatusType;
		Step : StepEnum;
	END_STRUCT;
	ControlCmdType : 	STRUCT
		StartCycle : BOOL;
	END_STRUCT;
	ControlParType : 	STRUCT
		CyclesToDo : INT;
	END_STRUCT;
	ControlStatusType : 	STRUCT
		ActPosition : LREAL;
		ActVelocity : REAL;
	END_STRUCT;
END_TYPE
```

### gProgramsVar.var
```iecst
VAR
	gControl : ControlTypeMain;
END_VAR
```

### Program Logical/Main/MainControl (IEC) - Main - control task

#### Auto.st - Init, cyclic, exit code
```iecst
PROGRAM _INIT
	(* Insert code here *)
END_PROGRAM

PROGRAM _CYCLIC
	(* Insert code here *)
	// do wyjebania tension enable
	actStopped;
	actStopping;
	actAborting;
	actAborted;
	actClearing;
	actProdResetting;
	actProdIdle;
	actProdStarting;
	actProdExecute;
	actProdCompleting;
	actProdComplete;
	actManResetting;
	actManIdle;

END_PROGRAM

PROGRAM _EXIT
	(* Insert code here *)

END_PROGRAM
```

#### lAutoType.typ - Local data types
```iecst
TYPE
	StoppedEnum :
		(
		STOPPED_IDLE (*STOPPED_IDLE*)
		);
	MainType : 	STRUCT
		PackMLStep : MainCmdType;
	END_STRUCT;
	MainCmdType : 	STRUCT
		Stopped : StoppedEnum;
	END_STRUCT;
END_TYPE
```

#### lAutoManualVar.var - Local variables
```iecst
VAR
	Main : MainType;
	xd : BOOL := TRUE;
	TESTbool : BOOL;
END_VAR
```

#### Package Logical/Main/MainControl/ActionsPackML - Actions for PackML

#### actStopped.st - STATE_STOPPED
```iecst
ACTION actStopped:
	IF MpPackMLStateIsActive(gPackMLCore, mpPACKML_STATE_STOPPED, PACKML_MODE_ALL) THEN

			gMainLogic.MotorMode.Production.Parameter.Velocity := 0.0;
			gMainLogic.MotorMode.Production.Parameter.Distance := 0.0;

			gMainLogic.MotorMode.Production.Cmd.Home := FALSE;
			gMainLogic.MotorMode.Production.Cmd.Reset := FALSE;

			gMainLogic.MotorMode.Production.Cmd.PowerOn := FALSE;

//			gMainLogic.MotorMode.Manual.Axis1.Cmd.PowerOn := FALSE;
//			gMainLogic.MotorMode.Manual.Axis2.Cmd.PowerOn := FALSE;
//			gMainLogic.MotorMode.Manual.Axis3.Cmd.PowerOn := FALSE;
//			gMainLogic.MotorMode.Manual.Axis1.Cmd.Enable := FALSE;
//			gMainLogic.MotorMode.Manual.Axis2.Cmd.Enable := FALSE;
//			gMainLogic.MotorMode.Manual.Axis3.Cmd.Enable := FALSE;

			// cala linia zeby ruszyc -> enable -> home -> power on -> start winding
	END_IF;
END_ACTION
```

#### actStopping.st - STATE_STOPPING
```iecst
ACTION actStopping:
// Free braking and transition to stopped
	IF MpPackMLStateIsActive(gPackMLCore, mpPACKML_STATE_STOPPING, PACKML_MODE_ALL) THEN
		gMainLogic.MotorMode.Production.Parameter.Distance := 0.0;
		gMainLogic.MotorMode.Production.Cmd.StartWinding := FALSE;
		gTensionLogic.Status.SetDancers := FALSE;
		gMainLogic.MotorMode.Production.Cmd.PowerOn := FALSE;
		gMainLogic.MotorMode.Production.Cmd.Reset := FALSE;
		gTensionLogic.Status.ProgressBarProcent := 0.0;

		//		gMainLogic.MotorMode.Manual.Axis1.Cmd.PowerOn := FALSE;
		//		gMainLogic.MotorMode.Manual.Axis2.Cmd.PowerOn := FALSE;
		//		gMainLogic.MotorMode.Manual.Axis3.Cmd.PowerOn := FALSE;
		IF NOT gTensionLogic.Status.LineIsPoweredOn THEN
			MpPackMLStateComplete(gPackMLCore, PACKML_MODE_ALL);
		END_IF;

	END_IF;
END_ACTION
```

#### actAborting.st - STATE_ABORTING
```iecst
ACTION actAborting:
// Everything stops (emergency/error stop)
	IF MpPackMLStateIsActive(gPackMLCore, mpPACKML_STATE_ABORTING, PACKML_MODE_ALL) THEN

		IF Status.ModeCurrent = 'Production' THEN
			gMainLogic.MotorMode.Production.Parameter.Velocity := 0.0;
			gMainLogic.MotorMode.Production.Cmd.StartWinding := FALSE;
			gTensionLogic.Status.ProgressBarProcent := 0.0;
			gMainLogic.MotorMode.Production.Cmd.Reset := TRUE;

			MpPackMLStateComplete(gPackMLCore, PACKML_MODE_ALL);
		END_IF;

		IF Status.ModeCurrent = 'Manual' THEN
			gMainLogic.MotorMode.Manual.Axis1.Cmd.JogAxis := FALSE;
			gMainLogic.MotorMode.Manual.Axis2.Cmd.JogAxis := FALSE;
			gMainLogic.MotorMode.Manual.Axis3.Cmd.JogAxis := FALSE;
			gMainLogic.MotorMode.Manual.JogWithTenReg := FALSE;

			MpPackMLStateComplete(gPackMLCore, PACKML_MODE_ALL);
		END_IF;

	END_IF;
END_ACTION
```

#### actAborted.st - STATE_ABORTED
```iecst
ACTION actAborted:
// Just pass to clearing
	IF MpPackMLStateIsActive(gPackMLCore, mpPACKML_STATE_ABORTED, PACKML_MODE_ALL) THEN
		IF NOT gHMI.Alarms.PendingAlarms THEN
			gMainLogic.MotorMode.Production.Cmd.Reset := FALSE;
	  		MpPackMLBasicUIConnect.StateControl.Clear := TRUE;
		END_IF;

	END_IF;
END_ACTION
```

#### actClearing.st - STATE_CLEARING
```iecst
ACTION actClearing:

	IF MpPackMLStateIsActive(gPackMLCore, mpPACKML_STATE_CLEARING, PACKML_MODE_ALL) THEN

		IF gHMI.Alarms.PendingAlarms THEN
			MpPackMLBasicUIConnect.StateControl.Abort := TRUE;
		ELSE
			MpPackMLStateComplete(gPackMLCore, PACKML_MODE_ALL);
		END_IF;

	END_IF;
END_ACTION
```

#### Package Logical/Main/MainControl/ActionsPackML/Manual - Actions specific to Manual mode

#### actManResetting.st - STATE_RESETTING [Manual]
```iecst
ACTION actManResetting:
// Nothing is powered, just go to IDLE
	IF MpPackMLStateIsActive(gPackMLCore, mpPACKML_STATE_RESETTING, PACKML_MODE_MANUAL) THEN

		// Completely disable all axes
		gMainLogic.MotorMode.Manual.Axis1.Cmd.PowerOn := FALSE;
		gMainLogic.MotorMode.Manual.Axis2.Cmd.PowerOn := FALSE;
		gMainLogic.MotorMode.Manual.Axis3.Cmd.PowerOn := FALSE;
		gMainLogic.MotorMode.Manual.Axis1.Cmd.Enable := FALSE;
		gMainLogic.MotorMode.Manual.Axis2.Cmd.Enable := FALSE;
		gMainLogic.MotorMode.Manual.Axis3.Cmd.Enable := FALSE;
		gMainLogic.MotorMode.Manual.JogWithTenReg := FALSE;

		// Go directly to IDLE
		MpPackMLStateComplete(gPackMLCore, PACKML_MODE_ALL);

	END_IF;
END_ACTION
```

#### actManIdle.st - STATE_IDLE [Manual]
```iecst
ACTION actManIdle:
// Everything can be done - individual axis jogging and tension regulation available
	IF MpPackMLStateIsActive(gPackMLCore, mpPACKML_STATE_IDLE, PACKML_MODE_MANUAL) THEN
		gHMI.Manual.JogLeftRight.Activate := gMainLogic.MotorMode.Production.Cmd.Home;
		gHMI.Manual.JogLeftRight.Activate := gMainLogic.MotorMode.Production.Cmd.PowerOn;

//		gHMI.

	END_IF;
END_ACTION
```

#### Package Logical/Main/MainControl/ActionsPackML/Production - Actions specific to Production mode

#### actProdResetting.st - STATE_RESETTING [Production]
```iecst
ACTION actProdResetting:
// Auto mode: start regulator (power axes) and turn off outputs
	IF MpPackMLStateIsActive(gPackMLCore, mpPACKML_STATE_RESETTING, PACKML_MODE_PRODUCTION) THEN

		gMainLogic.MotorMode.Production.Cmd.Reset := TRUE;
		gMainLogic.MotorMode.Production.Cmd.Home := TRUE;
		gMainLogic.MotorMode.Production.Cmd.PowerOn := TRUE;
		gMainLogic.MotorMode.Production.Parameter.Velocity := 0.0;
		gMainLogic.MotorMode.Production.Parameter.Distance := 0.0;

		IF gTensionLogic.Status.LineIsHomed AND
			gTensionLogic.Status.LineIsPoweredOn THEN

			gMainLogic.MotorMode.Production.Cmd.Home := FALSE;
			MpPackMLStateComplete(gPackMLCore, PACKML_MODE_PRODUCTION);
		END_IF;

	END_IF;
END_ACTION
```

#### actProdIdle.st - STATE_IDLE [Production]
```iecst
ACTION actProdIdle:
// Waiting for START button press
	IF MpPackMLStateIsActive(gPackMLCore, mpPACKML_STATE_IDLE, PACKML_MODE_PRODUCTION) THEN

		gMainLogic.MotorMode.Production.Cmd.Reset := FALSE;
		gMainLogic.MotorMode.Production.Parameter.Velocity := gHMI.Recipe.CurrentRecipe.Speed;
		gMainLogic.MotorMode.Production.Parameter.DancerPos1 := gHMI.Recipe.CurrentRecipe.TensionLeft;
		gMainLogic.MotorMode.Production.Parameter.DancerPos2 := gHMI.Recipe.CurrentRecipe.TensionRight;

		IF gHMI.Main.MaterialAdj.Direction THEN
			gMainLogic.MotorMode.Production.Parameter.Distance := gHMI.Main.MaterialAdj.Length;
		ELSE
			gMainLogic.MotorMode.Production.Parameter.Distance := -gHMI.Main.MaterialAdj.Length;
		END_IF;
		IF NOT gTensionLogic.Status.EnableAxis1 OR NOT gTensionLogic.Status.EnableAxis2 OR NOT gTensionLogic.Status.EnableAxis3 THEN
			MpPackMLBasicUIConnect.StateControl.Abort := TRUE;
		END_IF;
		IF NOT gTensionLogic.Status.ErrorExist THEN
	  		MpPackMLStateComplete(gPackMLCore, PACKML_MODE_PRODUCTION);
		END_IF;
	END_IF;
END_ACTION
```

#### actProdStarting.st - STATE_STARTING [Production]
```iecst
ACTION actProdStarting:
// Turn on tension regulator, achieve and maintain stable tension for 1s
	IF MpPackMLStateIsActive(gPackMLCore, mpPACKML_STATE_STARTING, PACKML_MODE_PRODUCTION) THEN

	gTensionLogic.Status.SetDancers := TRUE;
		IF NOT gTensionLogic.Status.EnableAxis1 OR NOT gTensionLogic.Status.EnableAxis2 OR NOT gTensionLogic.Status.EnableAxis3 THEN
			MpPackMLBasicUIConnect.StateControl.Abort := TRUE;
		END_IF;
		IF gMainLogic.MotorMode.Production.Status.TensionReady THEN
			MpPackMLStateComplete(gPackMLCore, PACKML_MODE_PRODUCTION);
		END_IF;

	END_IF;
END_ACTION
```

#### actProdExecute.st - STATE_EXECUTE [Production]
```iecst
ACTION actProdExecute:
// Wind material 0.9m, then go to completing
	IF MpPackMLStateIsActive(gPackMLCore, mpPACKML_STATE_EXECUTE, PACKML_MODE_PRODUCTION) THEN

		gMainLogic.MotorMode.Production.Cmd.StartWinding := TRUE;
		IF NOT gTensionLogic.Status.EnableAxis1 OR NOT gTensionLogic.Status.EnableAxis2 OR NOT gTensionLogic.Status.EnableAxis3 THEN
			MpPackMLBasicUIConnect.StateControl.Abort := TRUE;
		END_IF;
		IF gMainLogic.MotorMode.Production.Cmd.StartWinding THEN
			IF gTensionLogic.Status.MoveDone THEN
				gMainLogic.MotorMode.Production.Cmd.StartWinding := FALSE;
				MpPackMLStateComplete(gPackMLCore, PACKML_MODE_PRODUCTION);
			END_IF;
		END_IF;

	END_IF;
END_ACTION
```

#### actProdCompleting.st - STATE_COMPLETING [Production]
```iecst
ACTION actProdCompleting:
// Wait until reaches end and stop everything, go to complete
	IF MpPackMLStateIsActive(gPackMLCore, mpPACKML_STATE_COMPLETING, PACKML_MODE_PRODUCTION) THEN
		gMainLogic.MotorMode.Production.Cmd.StartWinding := FALSE;
		gMainLogic.MotorMode.Production.Parameter.Velocity := 0.0;
		IF NOT gTensionLogic.Status.EnableAxis1 OR NOT gTensionLogic.Status.EnableAxis2 OR NOT gTensionLogic.Status.EnableAxis3 THEN
			MpPackMLBasicUIConnect.StateControl.Abort := TRUE;
		END_IF;
		MpPackMLStateComplete(gPackMLCore, PACKML_MODE_PRODUCTION);
	END_IF;
END_ACTION
```

#### actProdComplete.st - STATE_COMPLETE [Production]
```iecst
ACTION actProdComplete:
// Clear variables
	IF MpPackMLStateIsActive(gPackMLCore, mpPACKML_STATE_COMPLETE, PACKML_MODE_PRODUCTION) THEN

		gMainLogic.MotorMode.Production.Parameter.Distance := 0.0;
		IF NOT gTensionLogic.Status.EnableAxis1 OR NOT gTensionLogic.Status.EnableAxis2 OR NOT gTensionLogic.Status.EnableAxis3 THEN
			MpPackMLBasicUIConnect.StateControl.Abort := TRUE;
		END_IF;
	END_IF;
END_ACTION
```

#### Constants.var
```iecst
VAR CONSTANT
	PACKML_MODE_ALL : USINT := 0;
END_VAR
```

### Constants.var - not listed in the package file held
```iecst
VAR CONSTANT
	PACKML_MODE_ALL: DINT := 0;
END_VAR
```

### Program Logical/Main/ActionsPackML

#### actAborted.st
```iecst
ACTION actAborted:
	// acknowlege all na liscie alarmow powoduje przejscie do clearing
END_ACTION
```

#### actAborting.st
```iecst
ACTION actAborting:
	// wszystko sie zatrzymuje
END_ACTION
```

#### actClearing.st
```iecst
ACTION actClearing:
	// acknowlege all na liscie alarmow

END_ACTION
```

#### actStopping.st
```iecst
ACTION actStopping:
	// wyhamowanie swobodne i przejscie do stopped

END_ACTION
```

- Visualisation Logical/mappView (not shown)

### gHmiVar.var
```iecst
VAR
	gHMI : HMI_type;
END_VAR
```

### gHmiTypes.typ
```iecst
(*Main type*)

TYPE
	HMI_type : 	STRUCT
		Recipe : Recipe_type;
		Manual : Manual_type;
		ControlBtn : ControlBtn_type;
		Charts : Charts_type;
		ModuleOK : ModuleOK_type;
		Main : MainPage_type;
		Alarms : Alarms_type;
		Data : Data_type;
	END_STRUCT;
END_TYPE

(*Main page*)

TYPE
	RollAdj_type : 	STRUCT
		Left : BOOL;
		Right : BOOL;
		LeftNum : REAL;
		RightNum : REAL;
	END_STRUCT;
	MainPage_type : 	STRUCT
		RollAdj : RollAdj_type;
		MaterialAdj : MaterialAdj_type;
	END_STRUCT;
	MaterialAdj_type : 	STRUCT
		Length : REAL;
		Direction : BOOL;
	END_STRUCT;
END_TYPE

(*Start, stop, reset, auto/manual buttons*)

TYPE
	ControlBtn_type : 	STRUCT
		Start : BOOL;
		Stop : BOOL;
		Reset : BOOL;
		AutoManual : BOOL;
	END_STRUCT;
END_TYPE

(*Recipe*)

TYPE
	DencerPI_type : 	STRUCT
		P : REAL;
		I : REAL;
	END_STRUCT;
	Recipe_type : 	STRUCT
		CurrentRecipe : CurrentRecipe_type;
		EnableEditing : BOOL;
		Load : BOOL;
	END_STRUCT;
	CurrentRecipe_type : 	STRUCT
		TensionLeft : REAL := 50.0; (* Naciąg lewy, zakres 0–14 cm *)
		TensionRight : REAL := 50.0; (* Naciąg prawy, zakres 0–14 cm *)
		Speed : REAL := 0.0; (* Prędkość taśmy w m/s *)
		RollLeft : MaxMinRollSize_type;
		RollRight : MaxMinRollSize_type;
		DataRegistration : BOOL := FALSE; (* Rejestracja danych: FALSE = wył., TRUE = wł. *)
		Dencer1PID : DencerPI_type;
		Dencer2PID : DencerPI_type;
	END_STRUCT;
	MaxMinRollSize_type : 	STRUCT
		MaxSize : REAL := 0.0;
		MinSize : REAL := 0.0;
	END_STRUCT;
END_TYPE

(*Manual page*)

TYPE
	Manual_type : 	STRUCT
		JogLeftRight : JogLeftRight_type;
		JogMotors : JogMotors_type;
	END_STRUCT;
	JogLeftRight_type : 	STRUCT
		Activate : BOOL;
		JogLeft : BOOL;
		JogRight : BOOL;
		SetBeltSpeed : REAL;
		JogLeftTemp : BOOL;
		JogRightTemp : BOOL;
		DenserLeft : REAL;
		DenserRight : REAL;
	END_STRUCT;
	JogMotors_type : 	STRUCT
		Motor1 : manMotor_type;
		Motor2 : manMotor_type;
		Motor3 : manMotor_type;
	END_STRUCT;
	manMotor_type : 	STRUCT
		Activate : BOOL;
		Home : BOOL;
		Speed : REAL;
		Left : BOOL;
		Right : BOOL;
	END_STRUCT;
END_TYPE

(*Charts*)

TYPE
	Record_type : 	STRUCT
		Dancer1 : BOOL;
		Dancer2 : BOOL;
		Axis1 : BOOL;
		Axis2 : BOOL;
		Axis3 : BOOL;
	END_STRUCT;
	Data_type : 	STRUCT
		isSaving : STRING[80];
	END_STRUCT;
	Charts_type : 	STRUCT
		Dancer1 : REAL;
		Dancer2 : REAL;
		Vtape : REAL;
		Axis1 : REAL;
		Axis2 : REAL;
		Axis3 : REAL;
		Record : Record_type;
	END_STRUCT;
END_TYPE

(*ModuleOk*)

TYPE
	ModuleOK_type : 	STRUCT
		PowerSupply : BOOL;
		AnalogInput : BOOL;
		SystemBusTransmitter : BOOL;
		ControlKeypad : BOOL;
	END_STRUCT;
END_TYPE

(*Alarms*)

TYPE
	Alarms_type : 	STRUCT
		PendingAlarms : BOOL;
	END_STRUCT;
END_TYPE
```

### Program Logical/HMI/ManualPage (IEC)

#### Types.typ
```iecst
TYPE
	HMIType : 	STRUCT
		ManualPage : ManualPageType;
	END_STRUCT;
	ManualPageType : 	STRUCT
		Buttons : ButtonsManual;
	END_STRUCT;
	ButtonsManual : 	STRUCT
		Mot1Active : BOOL;
		Mot2Active : BOOL;
		Mot3Active : BOOL;
		Strings : BtnManualStrings;
	END_STRUCT;
	BtnManualStrings : 	STRUCT
		ON : STRING[80];
		OFF : STRING[80];
		Btn1 : STRING[80];
		Btn2 : STRING[80];
		Btn3 : STRING[80];
	END_STRUCT;
END_TYPE
```

#### Variables.var
```iecst
VAR
	HMI : HMIType;
END_VAR
```

#### Main.st
```iecst
PROGRAM _INIT

END_PROGRAM

PROGRAM _CYCLIC

END_PROGRAM

PROGRAM _EXIT

END_PROGRAM
```

### Program Logical/HMI/RecipePage (IEC)

#### Main.st - Init, cyclic, exit code
```iecst
PROGRAM _INIT
	MpRecepieXml_0.Enable := TRUE;
	MpRecepieXml_0.MpLink := ADR(MpLinkRecipes);
	MpRecepieXml_0.DeviceName := ADR('RECIPE');

	MpRecipeRegPar_0.Enable := TRUE;
	MpRecipeRegPar_0.MpLink := ADR(MpLinkRecipes);
	MpRecipeRegPar_0.PVName := ADR('gHMI.Recipe.CurrentRecipe');

	MpRecipeUI_0.Enable := TRUE;
	MpRecipeUI_0.MpLink := ADR(MpLinkRecipes);
	MpRecipeUI_0.UIConnect := ADR(UIConnect);

	UIConnect.Recipe.Filter := '*.xml';
END_PROGRAM

PROGRAM _CYCLIC
	MpRecepieXml_0();
	MpRecipeRegPar_0();
	MpRecipeUI_0();
	actRecipeManage;

	RecipeControl.LoadRecipe := '';
	brsstrcat(ADR(RecipeControl.LoadRecipe), ADR('USER/'));
	brsstrcat(ADR(RecipeControl.LoadRecipe), ADR(MpRecepieXml_0.Info.LastLoadedRecipe));

	IF UIConnect.Recipe.List.SelectedIndex >=3 THEN
		RecipeControl.TableControl.Offset := UIConnect.Recipe.List.SelectedIndex - 3;
	ELSE
		RecipeControl.TableControl.Offset := 0;
	END_IF;

	actImageBinding;

	IF MpRecepieXml_0.Error THEN
		MpRecepieXml_0.ErrorReset := TRUE;
	ELSE
		MpRecepieXml_0.ErrorReset := FALSE;
	END_IF;

	IF MpRecipeRegPar_0.Error THEN
		MpRecipeRegPar_0.ErrorReset := TRUE;
	ELSE
		MpRecipeRegPar_0.ErrorReset := FALSE;
	END_IF;

	IF MpRecipeUI_0.Error THEN
		MpRecipeUI_0.ErrorReset := TRUE;
	ELSE
		MpRecipeUI_0.ErrorReset := FALSE;
	END_IF;
END_PROGRAM

PROGRAM _EXIT
	MpRecepieXml_0.Enable := FALSE;
	MpRecepieXml_0();
	MpRecipeRegPar_0.Enable := FALSE;
	MpRecipeRegPar_0();
	MpRecipeUI_0.Enable := FALSE;
	MpRecipeUI_0();
END_PROGRAM
```

#### Types.typ - Local data types
```iecst
TYPE
	TableControl_type : 	STRUCT
		Config : STRING[80] := '{"specRows": [{"from":11, "to":20, "visible":false}]}';
		Offset : UINT;
	END_STRUCT;
	Edit_type : 	STRUCT
		SaveRecipe : BOOL;
		DialogOpen : BOOL;
	END_STRUCT;
	RecipeControl_type : 	STRUCT
		Edit : Edit_type;
		LoadRecipe : STRING[80] := '0';
		TableControl : TableControl_type;
		Error : BOOL;
	END_STRUCT;
	ImageDirectory_type : 	STRUCT
		LeftArrow : STRING[80];
		RightArrow : STRING[80];
		On : STRING[80];
		Off : STRING[80];
		Current : CurrentImage_type;
	END_STRUCT;
	CurrentImage_type : 	STRUCT
		CurrentArrow : STRING[80];
		CurrentOnOff : STRING[80];
	END_STRUCT;
	RecipeCreateSteps :
		( (*Steps for creating recipes*)
		IDLE := 0, (*Idle State *)
		CREATE_1 := 10, (*Create coffee mappRegular*)
		DONE_1 := 11, (*mappRegular was created*)
		CREATE_2 := 20, (*Create coffee mappEspresso*)
		DONE_2 := 21, (*mappEspresso was created*)
		CREATE_3 := 30, (*Create coffee mappCappuccino*)
		DONE_3 := 31, (*mappCappuccino was created*)
		CREATE_4 := 40, (*Create coffee mappMilkCoffee*)
		DONE_4 := 41, (*mappMilkCoffee was created*)
		REFRESH := 42,
		LOAD := 43,
		ALL_DONE := 50 (*All recipes were created*)
		);
END_TYPE
```

#### Variables.var - Local variables
```iecst
VAR
	MaterialWidningEDITRecipe : CurrentRecipe_type;
	MpRecepieXml_0 : MpRecipeXml;
	MpRecipeRegPar_0 : MpRecipeRegPar;
	MpRecipeUI_0 : MpRecipeUI;
	UIConnect : MpRecipeUIConnectType;
	ImageDirectory : ImageDirectory_type;
	RecipeCreateStep : RecipeCreateSteps := IDLE; (*Internal variable for recipe creating state machine*)
	RecipeControl : RecipeControl_type;
END_VAR
```

#### ImageBinding.st
```iecst
ACTION actImageBinding:
	ImageDirectory.On := 'Media/SymbolLib/Symbols/Accept.svg';
	ImageDirectory.Off := 'Media/SymbolLib/Edit/Close.svg';

	IF gHMI.Recipe.CurrentRecipe.DataRegistration = TRUE THEN
		ImageDirectory.Current.CurrentOnOff := ImageDirectory.On;
	ELSE
		ImageDirectory.Current.CurrentOnOff := ImageDirectory.Off;
	END_IF;

END_ACTION
```
